// TIA Portal V19 export
FUNCTION_BLOCK "CoilHandling_FB"   // FB101, LAD
TITLE = COIL HANDLING MANAGER
// stored: MemoryReserve 100, SetENOAutomatically false
   VAR_INPUT
      AreaInterface : "AreaInterface";
      ZSI : "udt_ZoneSafetyInterface";
      DataIn : Struct
         PbMaterialBkw : Bool;
         PbMaterialFwd : Bool;
         PbExtraLowSpeed : Bool;
         SensorMatPresence_Decoiler : Bool;
         SensorMatPresence_StraightEntry : Bool;
         SensorMatPresence_StraightExit : Bool;
         SensorMatPresence_JBPinchExit : Bool;
         PbCoilReady : Bool;
         PbProvino : Bool;
         Decoiler2_PosizioneRazza : Bool;
      END_STRUCT;
      CIn : Struct
         DecoilersHRot : "DecoilersHRot_Status";
         Decoiler1 : "Decoiler_Status";
         Decoiler2 : "Decoiler_Status";
         Peeler : "Peeler_Status";
         Straigtener : "Straightener_Status";
         JB : "JB_Status";
         MaterialCounter : Struct
            AlrPresence : Bool;
            WngPresence : Bool;
            Data : "MatCountData";
         END_STRUCT;
         Loop : Struct
            SystemOn : Bool;
            Enable_FWD : Bool;
            Enable_BWD : Bool;
            SynchroRunning : Bool;
            MaxLength_Reeached : Bool;
            VelocityOverride : Real;
         END_STRUCT;
         Downstream : Struct
            Aut : Bool;
            MaterialPresence_Entry : Bool;
            MaterialPresence : Bool;
            LineVelocity : LReal;
         END_STRUCT;
         MES : "Prod_Coil_Ctrl";
      END_STRUCT;
      Config : "CoilHandling_Config";
      "ThicknessCheck_HW_ID_DL-PN" : HW_SUBMODULE := 784;
      ThicknessCheck_HW_ID_IL1000 : HW_SUBMODULE := 1042;
      ThicknessCheck_HW_ID_IL1050 : HW_SUBMODULE := 1043;
   END_VAR
   VAR_OUTPUT
      MachineInterface : "MachineInterface";
      COut : Struct
         Gen : Struct
            Material_STS : Int;   // 0=Empty; 1=Threading; 2= Full; 3= EOF Coil; 4= Separation
            MaterialPresence : Bool;
            MaterialMissing : Bool;
            NextEndOfMaterial : Bool;
            EmptyingConfirmed : Bool := FALSE;
            ExtraLowSpeedSelection : Bool;
            SemiAutomatic : Bool;
            Production_Running : Bool;
            DecoilerInLineNumber : Int;
            CoilDiameter : Real;
         END_STRUCT;
         DecoilersHRot : "DecoilersHRot_Manager";
         DecoilerInLine : "Decoiler_Manager";
         DecoilerOutLine : "Decoiler_Manager";
         Decoiler1 : "Decoiler_Manager";
         Decoiler2 : "Decoiler_Manager";
         Peeler : "Peeler_Manager";
         Straightener : "Straightener_Manager";
         JB : "JB_Manager";
         Loop : Struct
            Stop : Bool;
            Synchro_Request : Bool;
            MaterialMiddlePos_Request : Bool;
         END_STRUCT;
         MES : Struct
            Deroga_Spessore_Errato { ExternalWritable := 'False'} : Bool;
            Spessore_Lamiera_Errato { ExternalWritable := 'False'} : Bool;
            Spessore_Lamiera_Sensore_Valore : Real;
            Spessore_Lamiera_Errore_Valore { ExternalWritable := 'False'} : Real;
            Provino_Eseguito : Bool;
         END_STRUCT;
      END_STRUCT;
      DataOut : Struct
         Lamp_CoilReady : Bool;
         Lamp_ExtraLowSpeed : Bool;
         Lamp_Provino : Bool;
      END_STRUCT;
   END_VAR
   VAR_IN_OUT
      Pers : "CoilHandling_Persistent";
   END_VAR
   VAR
      Alarm : Struct
         MaterialMissing : Bool;
         S_MatPresence_StraightExit_NotOFF : Bool;
         MatCounterAlrPresence : Bool;
         EndOfMaterial : Bool;
         TichnessCheck { ExternalAccessible := 'False'; ExternalVisible := 'False'; ExternalWritable := 'False'} : Struct
            Err_Sensor_Get_PN_IO : Bool;
            Err_Sensor_Rack : Bool;
            Err_Sensor_Value : Bool;
            ThicknessOutOfRange : Bool;
         END_STRUCT;
         MES : Struct
            STOP_Provino { ExternalAccessible := 'False'; ExternalVisible := 'False'; ExternalWritable := 'False'} : Bool;
            STOP_Taglio_Fine_Ordini { ExternalAccessible := 'False'; ExternalVisible := 'False'; ExternalWritable := 'False'} : Bool;
            STOP_Manca_Dati_AspoInLinea { ExternalAccessible := 'False'; ExternalVisible := 'False'; ExternalWritable := 'False'} : Bool;
            STOP_FineTurno { ExternalAccessible := 'False'; ExternalVisible := 'False'; ExternalWritable := 'False'} : Bool;
            STOP_ControlloQualita { ExternalAccessible := 'False'; ExternalVisible := 'False'; ExternalWritable := 'False'} : Bool;
         END_STRUCT;
      END_STRUCT;
      Warning : Struct
         NotAutReady : Bool;
         MatCounterWngPresence : Bool;
         EmptyingIsON : Bool := FALSE;
         EndOfMaterial_StraightenetEntry : Bool;
         EndOfMaterial_StraightenetExit : Bool;
         EndOfCoilSequenceRunning : Bool;
         ExtraLowSpeedIsON : Bool;
         Decoiler2_RazzaNonInPosizione : Bool;
         StopInactivity : Bool;
         ThicnessCheck { ExternalAccessible := 'False'; ExternalVisible := 'False'; ExternalWritable := 'False'} : Struct
            SensorDisable : Bool;
            ThicknessOutOfRange : Bool;
            Err_Bypass : Bool;
         END_STRUCT;
         MES : Struct
            STOP_Manca_Dati_AspoInCarico : Bool;
         END_STRUCT;
      END_STRUCT;
      HMI : Struct
         B_ConfirmEmptying { ExternalAccessible := 'False'; ExternalVisible := 'False'; ExternalWritable := 'False'} : Bool;
         B_ConfirmEmptyingShow { ExternalAccessible := 'False'; ExternalVisible := 'False'; ExternalWritable := 'False'} : Bool;
         B_ConfirmEmptyingStatus : Bool;
         ThicknessControl : Struct
            Button_Exception : Bool;
            Button_Init : Bool;
            STATUS : Int;
         END_STRUCT;
      END_STRUCT;
      Ctrl : Struct
         Pause : Bool;
         Stop : Bool;
         Semiautomatic_MaterialFwd : Bool;
         Semiautomatic_MaterialBkw : Bool;
         EndOfCoil : Struct
            StraightRollEntry_Open : Bool;
            StraightRollExit_Open : Bool;
            StraightRollEntry_Close : Bool;
            StraightRollExit_Close : Bool;
            Straightener_Bwd : Bool;
            Straightener_Fwd : Bool;
            JB_Pinch_Open : Bool;
            JB_Pinch_Close : Bool;
            JB_Pinch_Fwd : Bool;
            JB_Cut_Rest : Bool;
            JB_Cut_Work : Bool;
            JB_Welder_Open : Bool;
            TargetPosMat_StraightEmpty : LReal;
            TargetPosMat_TailCutExe : LReal;
            TargetPosMat_JunctionExe : LReal;
            ChangeCoilExe : Bool;
            Decoiler_Fwd : Bool;
         END_STRUCT;
      END_STRUCT;
      Sts : Struct
         FeedStandstill : Bool;
         AlarmsPresence : Bool;
         WarningsPresence : Bool;
         EnableCycleStopProgrammed : Bool;
         MaterialFwdEnable : Bool;
         MaterialBkwEnable : Bool;
         CumulativeMaterialFwdRequest : Bool;
         Semiautomatic : Bool;
         ExtraLowSpeedSelectionPB : Bool;
         ExtraLowSpeedSelection : Bool;
         STOP_Feed_by_MES : Bool;
         STOP_CoilChange_By_MES : Bool;
         STOP_Inactivity : Bool;
         DecoilerInLine : "Decoiler_Status";
         DecoilerOutOfLine : "Decoiler_Status";
         EndOfCoil : Struct
            Status : Int;
            Cnd : Bool;
            Idle : Bool;
            EndOfSequence : Bool;
            PinchRoll_SpaceToStop : LReal;
            PosMat_AtEndMatPresence_StraightEnty : LReal;
            PosMat_AtEndMatPresence_StraightExit : LReal;
            MissingTargetPosMat_StraightEmpty : LReal;
            MissingToTargetPosMat_TailCutExe : LReal;
            StopPinchRoll_TargetPosMat_TailCutExe : Bool;
            Reached_TargetPosMat_TailCutExe : Bool;
            MissingToTargetPosMat_JunctionExe : LReal;
            StopPinchRoll_TargetPosMat_JunctionExe : Bool;
            Reached_TargetPosMat_JunctionExe : Bool;
         END_STRUCT;
         LoopSynchro : Struct
            Phase1_A : Bool;   // Coil diameter < limit
            Phase2_A : Bool;   // Mem synchro done
            Phase1_B : Bool;   // Coil diameter < limit
            Phase2_B : Bool;   // Mem synchro done
         END_STRUCT;
         MaterialMoveSemiAut : Struct
            Bwd_Phase1 : Bool;   // Move no feeding machine to rest
            Bwd_Phase1Cnd : Bool;
            Bwd_Phase2 : Bool;   // Move velocity = 0
            Bwd_Phase2Cnd : Bool;
            Bwd_Phase3 : Bool;   // Move velocity > 0
            Fwd_Phase1 : Bool;   // Move no feeding machine to rest
            Fwd_Phase1Cnd : Bool;
            Fwd_Phase2 : Bool;   // Move velocity = 0
            Fwd_Phase2Cnd : Bool;
            Fwd_Phase3 : Bool;   // Move velocity > 0
         END_STRUCT;
         MaterialMoveAut : Struct
            Fwd_Phase1 : Bool;   // Move no feeding machine to rest
            Fwd_Phase1Cnd : Bool;
            Fwd_Phase2 : Bool;   // Move velocity = 0
            Fwd_Phase2Cnd : Bool;
            Fwd_Phase3 : Bool;   // Move velocity > 0
         END_STRUCT;
      END_STRUCT;
      MatPresence_Decoiler : "DelayOnOff_R";
      MatPresence_StraightEntry : "DelayOnOff_R";
      MatPresence_StraightExit : "DelayOnOff_R";
      MatPresence_JBPinchExit : "DelayOnOff_R";
      Coil_LooseWrap : "CoilCheckLooseWrap";
      ThicknessCheck { S7_SetPoint := 'True'} : "ThicknessCheck_FB";
      CoilHandling_MES { S7_SetPoint := 'True'} : "CoilHandling_MES_FB";
      TON_Emptying : TON_TIME;
      TON_DecoilerNotMovingBkw : TON_TIME;
      TON_PinchrollFwd : TON_TIME;
      TON_StraightnerBwd : TON_TIME;
      TON_StraightnerFwd : TON_TIME;
      TON_SemiautoOFF : TON_TIME;
      TON_AutDisableAxes : TON_TIME;
      TON_StopInactivity : TON_TIME;
      AUX : Struct
         S_MatPresence_StraightEntry : Bool;
         S_MatPresence_StraightExit : Bool;
         PbMaterialFwd : Bool;
         PbMaterialBkw : Bool;
         PbExtraLowSpeed : Bool;
         ButtonForceLoopMiddle : Bool;
         PbCoilLoaded : Bool;
         StopLoop { ExternalAccessible := 'False'; ExternalVisible := 'False'; ExternalWritable := 'False'} : Bool;
      END_STRUCT;
   END_VAR
   VAR_TEMP
      PE : Struct
         Not_S_MatPresence_StraightEntry : Bool;
         Not_S_MatPresence_StraightExit : Bool;
         PbMaterialBkw : Bool;
         PbMaterialFwd : Bool;
         PbExtraLowSpeed : Bool;
      END_STRUCT;
      Req : Bool;
      Set : Bool;
      Rst : Bool;
      Cnd : Bool;
      Min : Bool;
      Max : Bool;
      OK : Bool;
      StraightRollEntry_Used : Bool;
      StraightRollExit_Used : Bool;
      DistanceSensorEntryExitStraight : LReal;
      DistanceLimit : LReal;
      LineVel : LReal;
      Decoiler_VelFactor : LReal;
      Straightener_VelFactor : LReal;
      OverRide_VelFactor : LReal;
      OverRide_VelFactor_Candidate : LReal;
      Delta : LReal;
      Vel : LReal;
      EnableStopInPhase : Bool;
      EnableStopProgrammed : Bool;
      EnableStopDoorOpeningReq : Bool;
      Set_1 : Bool;
      Rst_1 : Bool;
      Set_2 : Bool;
      Rst_2 : Bool;
      CaseA : Bool;
      CaseB : Bool;
      Empty : Bool;
      JunctionDone : Bool;
   END_VAR
   // MachineInterface.AutReady := TRUE;
   // MachineInterface.Aborting := FALSE;
   // MachineInterface.AckStopInPhase := FALSE;
   // MachineInterface.AckStopProgrammed := FALSE;
   // MachineInterface.MotionsStandStill := TRUE;
   // MachineInterface.AlarmsPresence := FALSE;
   // MachineInterface.WarningPresence := TRUE;
   VAR_TEMP   // added for the SCL form of the ladder/FBD networks
      _w1 : Bool;
      _w2 : Bool;
      _w3 : Bool;
   END_VAR
BEGIN

REGION Network 1 (SCL): Reset alarms
   IF #AreaInterface.RstAlarms THEN

       #Alarm.MaterialMissing := FALSE;
       #Alarm.S_MatPresence_StraightExit_NotOFF := FALSE;
       #Alarm.EndOfMaterial := FALSE;


       #Warning.Decoiler2_RazzaNonInPosizione := FALSE;
       #Warning.NotAutReady := FALSE;

   END_IF;
END_REGION

REGION Network 2: >
END_REGION

REGION Network 3: >
END_REGION

REGION Network 4: Straightenetr rolls entry / exit to use
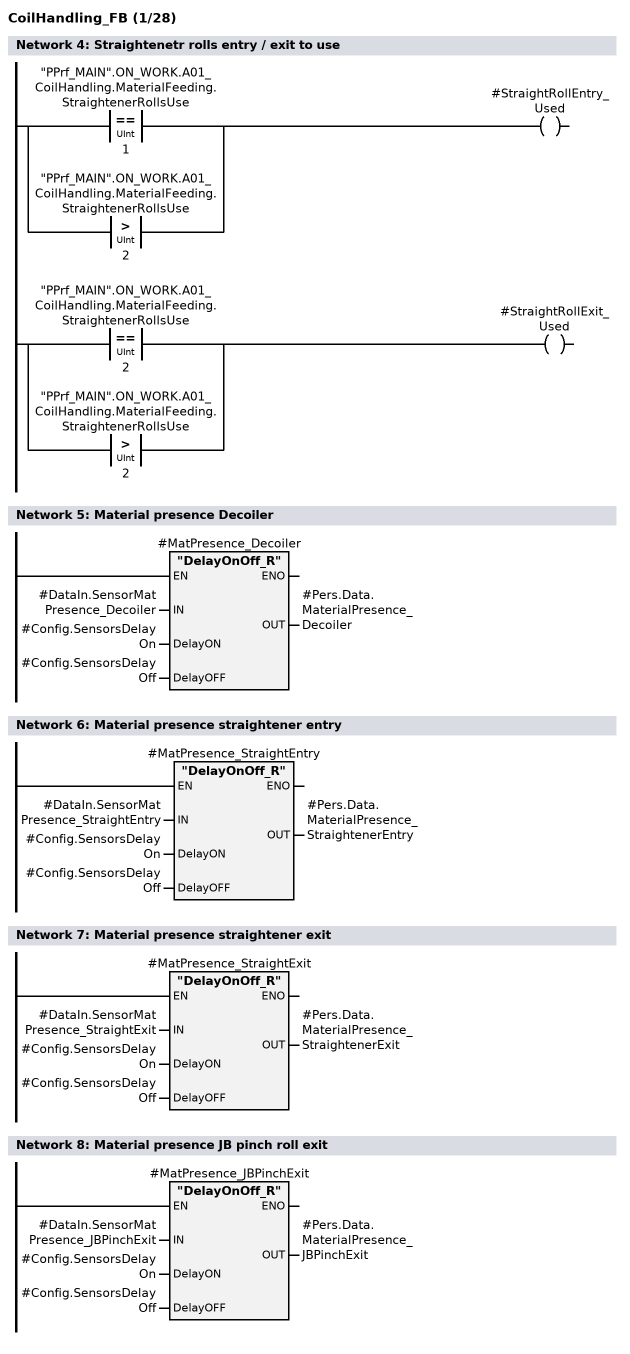
   RUNG wire#powerrail
      { S7_Templates := "SrcType := UInt" } EQ_Contact(in1 := "PPrf_MAIN".ON_WORK.A01_CoilHandling.MaterialFeeding.StraightenerRollsUse, in2 := 1)
      wire#w1
      Coil( #StraightRollEntry_Used )
   END_RUNG
   RUNG wire#powerrail
      { S7_Templates := "SrcType := UInt" } GT_Contact(in1 := "PPrf_MAIN".ON_WORK.A01_CoilHandling.MaterialFeeding.StraightenerRollsUse, in2 := 2)
   END_RUNG wire#w1
   RUNG wire#powerrail
      { S7_Templates := "SrcType := UInt" } EQ_Contact(in1 := "PPrf_MAIN".ON_WORK.A01_CoilHandling.MaterialFeeding.StraightenerRollsUse, in2 := 2)
      wire#w2
      Coil( #StraightRollExit_Used )
   END_RUNG
   RUNG wire#powerrail
      { S7_Templates := "SrcType := UInt" } GT_Contact(in1 := "PPrf_MAIN".ON_WORK.A01_CoilHandling.MaterialFeeding.StraightenerRollsUse, in2 := 2)
   END_RUNG wire#w2
   // the same network as SCL:
   #StraightRollEntry_Used := ("PPrf_MAIN".ON_WORK.A01_CoilHandling.MaterialFeeding.StraightenerRollsUse = 1) OR ("PPrf_MAIN".ON_WORK.A01_CoilHandling.MaterialFeeding.StraightenerRollsUse > 2);
   #StraightRollExit_Used := ("PPrf_MAIN".ON_WORK.A01_CoilHandling.MaterialFeeding.StraightenerRollsUse = 2) OR ("PPrf_MAIN".ON_WORK.A01_CoilHandling.MaterialFeeding.StraightenerRollsUse > 2);
END_REGION

REGION Network 5: Material presence Decoiler
   RUNG wire#powerrail
      #MatPresence_Decoiler(IN := #DataIn.SensorMatPresence_Decoiler, DelayON := #Config.SensorsDelayOn, DelayOFF := #Config.SensorsDelayOff, OUT => #Pers.Data.MaterialPresence_Decoiler)
   END_RUNG
   // the same network as SCL:
   #MatPresence_Decoiler(IN := #DataIn.SensorMatPresence_Decoiler,   // "DelayOnOff_R"
                         DelayON := #Config.SensorsDelayOn,
                         DelayOFF := #Config.SensorsDelayOff,
                         OUT => #Pers.Data.MaterialPresence_Decoiler);
END_REGION

REGION Network 6: Material presence straightener entry
   RUNG wire#powerrail
      #MatPresence_StraightEntry(IN := #DataIn.SensorMatPresence_StraightEntry, DelayON := #Config.SensorsDelayOn, DelayOFF := #Config.SensorsDelayOff, OUT => #Pers.Data.MaterialPresence_StraightenerEntry)
   END_RUNG
   // the same network as SCL:
   #MatPresence_StraightEntry(IN := #DataIn.SensorMatPresence_StraightEntry,   // "DelayOnOff_R"
                           DelayON := #Config.SensorsDelayOn,
                           DelayOFF := #Config.SensorsDelayOff,
                           OUT => #Pers.Data.MaterialPresence_StraightenerEntry);
END_REGION

REGION Network 7: Material presence straightener exit
   RUNG wire#powerrail
      #MatPresence_StraightExit(IN := #DataIn.SensorMatPresence_StraightExit, DelayON := #Config.SensorsDelayOn, DelayOFF := #Config.SensorsDelayOff, OUT => #Pers.Data.MaterialPresence_StraightenerExit)
   END_RUNG
   // the same network as SCL:
   #MatPresence_StraightExit(IN := #DataIn.SensorMatPresence_StraightExit,   // "DelayOnOff_R"
                           DelayON := #Config.SensorsDelayOn,
                           DelayOFF := #Config.SensorsDelayOff,
                           OUT => #Pers.Data.MaterialPresence_StraightenerExit);
END_REGION

REGION Network 8: Material presence JB pinch roll exit
   RUNG wire#powerrail
      #MatPresence_JBPinchExit(IN := #DataIn.SensorMatPresence_JBPinchExit, DelayON := #Config.SensorsDelayOn, DelayOFF := #Config.SensorsDelayOff, OUT => #Pers.Data.MaterialPresence_JBPinchExit)
   END_RUNG
   // the same network as SCL:
   #MatPresence_JBPinchExit(IN := #DataIn.SensorMatPresence_JBPinchExit,   // "DelayOnOff_R"
                           DelayON := #Config.SensorsDelayOn,
                           DelayOFF := #Config.SensorsDelayOff,
                           OUT => #Pers.Data.MaterialPresence_JBPinchExit);
END_REGION

REGION Network 9: >
END_REGION

REGION Network 10: >
END_REGION

REGION Network 11: Material junction done
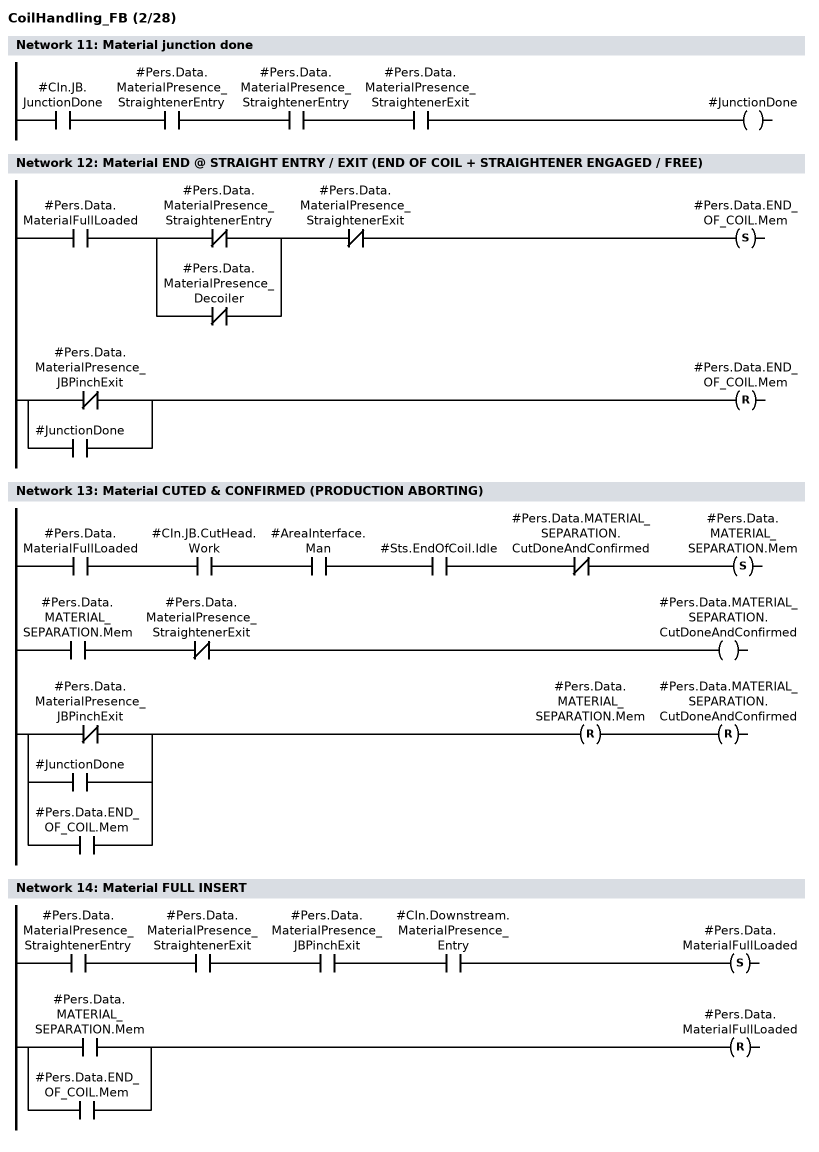
   RUNG wire#powerrail
      Contact( #CIn.JB.JunctionDone )
      Contact( #Pers.Data.MaterialPresence_StraightenerEntry )
      Contact( #Pers.Data.MaterialPresence_StraightenerEntry )
      Contact( #Pers.Data.MaterialPresence_StraightenerExit )
      Coil( #JunctionDone )
   END_RUNG
   // the same network as SCL:
   #JunctionDone := #CIn.JB.JunctionDone AND #Pers.Data.MaterialPresence_StraightenerEntry AND #Pers.Data.MaterialPresence_StraightenerEntry AND #Pers.Data.MaterialPresence_StraightenerExit;
END_REGION

REGION Network 12: Material END @ STRAIGHT ENTRY / EXIT (END OF COIL + STRAIGHTENER ENGAGED / FREE)
   RUNG wire#powerrail
      Contact( #Pers.Data.MaterialFullLoaded )
      wire#w1
      I_Contact( #Pers.Data.MaterialPresence_StraightenerEntry )
      wire#w2
      I_Contact( #Pers.Data.MaterialPresence_StraightenerExit )
      S_Coil( #Pers.Data.END_OF_COIL.Mem )
   END_RUNG
   RUNG wire#w1
      I_Contact( #Pers.Data.MaterialPresence_Decoiler )
   END_RUNG wire#w2
   RUNG wire#powerrail
      I_Contact( #Pers.Data.MaterialPresence_JBPinchExit )
      wire#w3
      R_Coil( #Pers.Data.END_OF_COIL.Mem )
   END_RUNG
   RUNG wire#powerrail
      Contact( #JunctionDone )
   END_RUNG wire#w3
   // the same network as SCL:
   IF #Pers.Data.MaterialFullLoaded AND (NOT #Pers.Data.MaterialPresence_StraightenerEntry OR NOT #Pers.Data.MaterialPresence_Decoiler) AND NOT #Pers.Data.MaterialPresence_StraightenerExit THEN
       #Pers.Data.END_OF_COIL.Mem := TRUE;
   END_IF;
   IF NOT #Pers.Data.MaterialPresence_JBPinchExit OR #JunctionDone THEN
       #Pers.Data.END_OF_COIL.Mem := FALSE;
   END_IF;
END_REGION

REGION Network 13: Material CUTED & CONFIRMED (PRODUCTION ABORTING)
   RUNG wire#powerrail
      Contact( #Pers.Data.MaterialFullLoaded )
      Contact( #CIn.JB.CutHead.Work )
      Contact( #AreaInterface.Man )
      Contact( #Sts.EndOfCoil.Idle )
      I_Contact( #Pers.Data.MATERIAL_SEPARATION.CutDoneAndConfirmed )
      S_Coil( #Pers.Data.MATERIAL_SEPARATION.Mem )
   END_RUNG
   RUNG wire#powerrail
      Contact( #Pers.Data.MATERIAL_SEPARATION.Mem )
      I_Contact( #Pers.Data.MaterialPresence_StraightenerExit )
      Coil( #Pers.Data.MATERIAL_SEPARATION.CutDoneAndConfirmed )
   END_RUNG
   RUNG wire#powerrail
      I_Contact( #Pers.Data.MaterialPresence_JBPinchExit )
      wire#w1
      R_Coil( #Pers.Data.MATERIAL_SEPARATION.Mem )
      R_Coil( #Pers.Data.MATERIAL_SEPARATION.CutDoneAndConfirmed )
   END_RUNG
   RUNG wire#powerrail
      Contact( #JunctionDone )
   END_RUNG wire#w1
   RUNG wire#powerrail
      Contact( #Pers.Data.END_OF_COIL.Mem )
   END_RUNG wire#w1
   // the same network as SCL:
   IF #Pers.Data.MaterialFullLoaded AND #CIn.JB.CutHead.Work AND #AreaInterface.Man AND #Sts.EndOfCoil.Idle AND NOT #Pers.Data.MATERIAL_SEPARATION.CutDoneAndConfirmed THEN
       #Pers.Data.MATERIAL_SEPARATION.Mem := TRUE;
   END_IF;
   #Pers.Data.MATERIAL_SEPARATION.CutDoneAndConfirmed := #Pers.Data.MATERIAL_SEPARATION.Mem AND NOT #Pers.Data.MaterialPresence_StraightenerExit;
   IF NOT #Pers.Data.MaterialPresence_JBPinchExit OR #JunctionDone OR #Pers.Data.END_OF_COIL.Mem THEN
       #Pers.Data.MATERIAL_SEPARATION.Mem := FALSE;
       #Pers.Data.MATERIAL_SEPARATION.CutDoneAndConfirmed := FALSE;
   END_IF;
END_REGION

REGION Network 14: Material FULL INSERT
   RUNG wire#powerrail
      Contact( #Pers.Data.MaterialPresence_StraightenerEntry )
      Contact( #Pers.Data.MaterialPresence_StraightenerExit )
      Contact( #Pers.Data.MaterialPresence_JBPinchExit )
      Contact( #CIn.Downstream.MaterialPresence_Entry )
      S_Coil( #Pers.Data.MaterialFullLoaded )
   END_RUNG
   RUNG wire#powerrail
      Contact( #Pers.Data.MATERIAL_SEPARATION.Mem )
      wire#w1
      R_Coil( #Pers.Data.MaterialFullLoaded )
   END_RUNG
   RUNG wire#powerrail
      Contact( #Pers.Data.END_OF_COIL.Mem )
   END_RUNG wire#w1
   // the same network as SCL:
   IF #Pers.Data.MaterialPresence_StraightenerEntry AND #Pers.Data.MaterialPresence_StraightenerExit AND #Pers.Data.MaterialPresence_JBPinchExit AND #CIn.Downstream.MaterialPresence_Entry THEN
       #Pers.Data.MaterialFullLoaded := TRUE;
   END_IF;
   IF #Pers.Data.MATERIAL_SEPARATION.Mem OR #Pers.Data.END_OF_COIL.Mem THEN
       #Pers.Data.MaterialFullLoaded := FALSE;
   END_IF;
END_REGION

REGION Network 15: Material presence for keep running the material even thoug is not full insterted
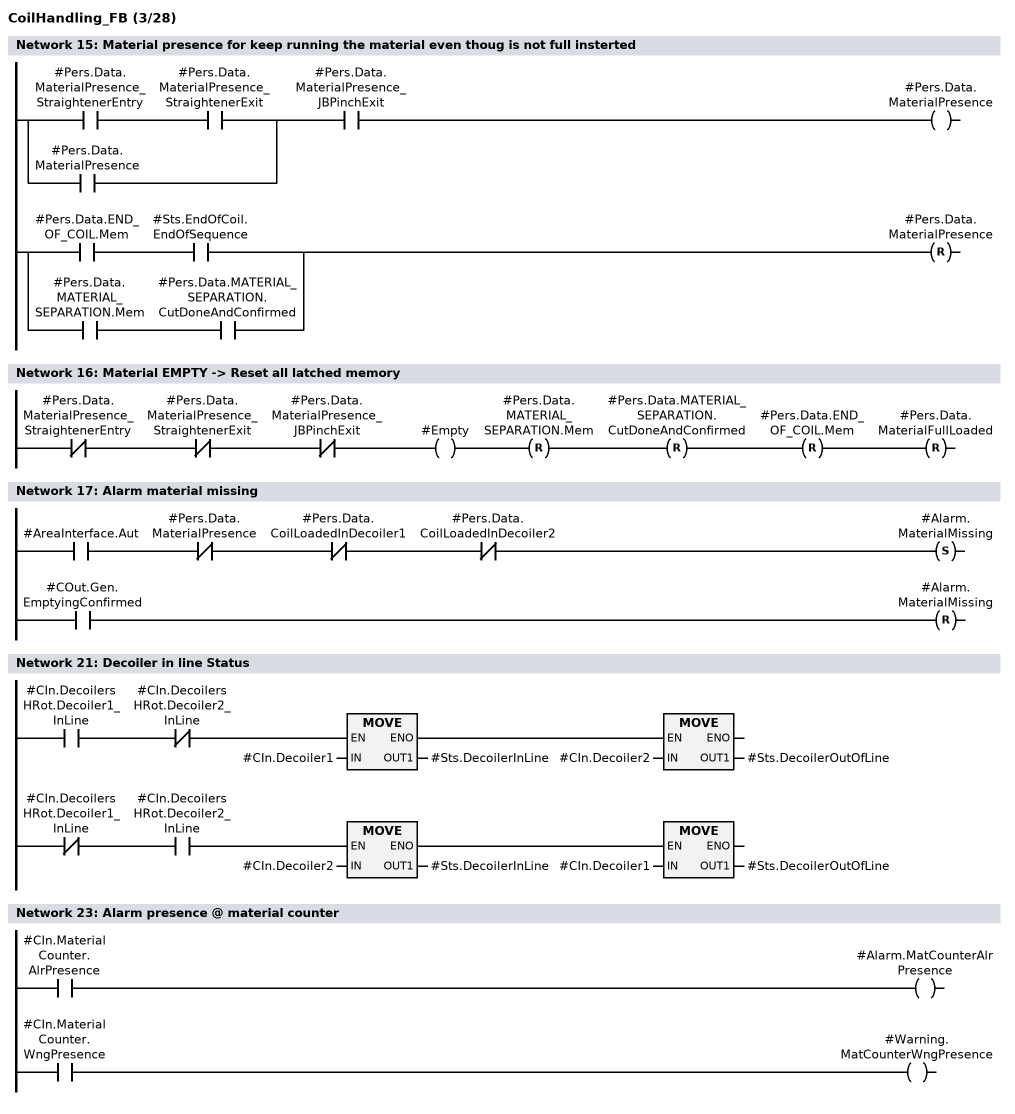
   RUNG wire#powerrail
      Contact( #Pers.Data.MaterialPresence_StraightenerEntry )
      Contact( #Pers.Data.MaterialPresence_StraightenerExit )
      wire#w1
      Contact( #Pers.Data.MaterialPresence_JBPinchExit )
      Coil( #Pers.Data.MaterialPresence )
   END_RUNG
   RUNG wire#powerrail
      Contact( #Pers.Data.MaterialPresence )
   END_RUNG wire#w1
   RUNG wire#powerrail
      Contact( #Pers.Data.END_OF_COIL.Mem )
      Contact( #Sts.EndOfCoil.EndOfSequence )
      wire#w2
      R_Coil( #Pers.Data.MaterialPresence )
   END_RUNG
   RUNG wire#powerrail
      Contact( #Pers.Data.MATERIAL_SEPARATION.Mem )
      Contact( #Pers.Data.MATERIAL_SEPARATION.CutDoneAndConfirmed )
   END_RUNG wire#w2
   // the same network as SCL:
   #Pers.Data.MaterialPresence := ((#Pers.Data.MaterialPresence_StraightenerEntry AND #Pers.Data.MaterialPresence_StraightenerExit) OR #Pers.Data.MaterialPresence) AND #Pers.Data.MaterialPresence_JBPinchExit;
   IF (#Pers.Data.END_OF_COIL.Mem AND #Sts.EndOfCoil.EndOfSequence) OR (#Pers.Data.MATERIAL_SEPARATION.Mem AND #Pers.Data.MATERIAL_SEPARATION.CutDoneAndConfirmed) THEN
       #Pers.Data.MaterialPresence := FALSE;
   END_IF;
END_REGION

REGION Network 16: Material EMPTY -> Reset all latched memory
   RUNG wire#powerrail
      I_Contact( #Pers.Data.MaterialPresence_StraightenerEntry )
      I_Contact( #Pers.Data.MaterialPresence_StraightenerExit )
      I_Contact( #Pers.Data.MaterialPresence_JBPinchExit )
      Coil( #Empty )
      R_Coil( #Pers.Data.MATERIAL_SEPARATION.Mem )
      R_Coil( #Pers.Data.MATERIAL_SEPARATION.CutDoneAndConfirmed )
      R_Coil( #Pers.Data.END_OF_COIL.Mem )
      R_Coil( #Pers.Data.MaterialFullLoaded )
   END_RUNG
   // the same network as SCL:
   #Empty := NOT #Pers.Data.MaterialPresence_StraightenerEntry AND NOT #Pers.Data.MaterialPresence_StraightenerExit AND NOT #Pers.Data.MaterialPresence_JBPinchExit;
   IF #Empty THEN
       #Pers.Data.MATERIAL_SEPARATION.Mem := FALSE;
       #Pers.Data.MATERIAL_SEPARATION.CutDoneAndConfirmed := FALSE;
       #Pers.Data.END_OF_COIL.Mem := FALSE;
       #Pers.Data.MaterialFullLoaded := FALSE;
   END_IF;
END_REGION

REGION Network 17: Alarm material missing
   RUNG wire#powerrail
      Contact( #AreaInterface.Aut )
      I_Contact( #Pers.Data.MaterialPresence )
      I_Contact( #Pers.Data.CoilLoadedInDecoiler1 )
      I_Contact( #Pers.Data.CoilLoadedInDecoiler2 )
      S_Coil( #Alarm.MaterialMissing )
   END_RUNG
   RUNG wire#powerrail
      Contact( #COut.Gen.EmptyingConfirmed )
      R_Coil( #Alarm.MaterialMissing )
   END_RUNG
   // the same network as SCL:
   IF #AreaInterface.Aut AND NOT #Pers.Data.MaterialPresence AND NOT #Pers.Data.CoilLoadedInDecoiler1 AND NOT #Pers.Data.CoilLoadedInDecoiler2 THEN
       #Alarm.MaterialMissing := TRUE;
   END_IF;
   IF #COut.Gen.EmptyingConfirmed THEN #Alarm.MaterialMissing := FALSE; END_IF;
END_REGION

REGION Network 18: >
END_REGION

REGION Network 19 (SCL): Material status
   IF #Empty
   THEN
       #COut.Gen.Material_STS := "MAT_EMPTY";
   ELSIF #Pers.Data.END_OF_COIL.Mem
   THEN
       #COut.Gen.Material_STS := "MAT_EOF_COIL";
   ELSIF #Pers.Data.MATERIAL_SEPARATION.Mem
   THEN
       #COut.Gen.Material_STS := "MAT_SPERATION";

   ELSIF #Pers.Data.MaterialFullLoaded
   THEN
       #COut.Gen.Material_STS := "MAT_FULL";
   ELSE
       #COut.Gen.Material_STS := "MAT_INTRODUCTION";
   END_IF;
END_REGION

REGION Network 20: >
END_REGION

REGION Network 21: Decoiler in line Status
   RUNG wire#powerrail
      Contact( #CIn.DecoilersHRot.Decoiler1_InLine )
      I_Contact( #CIn.DecoilersHRot.Decoiler2_InLine )
      Move(in := #CIn.Decoiler1, out1 => #Sts.DecoilerInLine)
      Move(in := #CIn.Decoiler2, out1 => #Sts.DecoilerOutOfLine)
   END_RUNG
   RUNG wire#powerrail
      I_Contact( #CIn.DecoilersHRot.Decoiler1_InLine )
      Contact( #CIn.DecoilersHRot.Decoiler2_InLine )
      Move(in := #CIn.Decoiler2, out1 => #Sts.DecoilerInLine)
      Move(in := #CIn.Decoiler1, out1 => #Sts.DecoilerOutOfLine)
   END_RUNG
   // the same network as SCL:
   IF #CIn.DecoilersHRot.Decoiler1_InLine AND NOT #CIn.DecoilersHRot.Decoiler2_InLine THEN
       #Sts.DecoilerInLine := #CIn.Decoiler1;
       #Sts.DecoilerOutOfLine := #CIn.Decoiler2;
   END_IF;
   IF NOT #CIn.DecoilersHRot.Decoiler1_InLine AND #CIn.DecoilersHRot.Decoiler2_InLine THEN
       #Sts.DecoilerInLine := #CIn.Decoiler2;
       #Sts.DecoilerOutOfLine := #CIn.Decoiler1;
   END_IF;
END_REGION

REGION Network 22: >
END_REGION

REGION Network 23: Alarm presence @ material counter
   RUNG wire#powerrail
      Contact( #CIn.MaterialCounter.AlrPresence )
      Coil( #Alarm.MatCounterAlrPresence )
   END_RUNG
   RUNG wire#powerrail
      Contact( #CIn.MaterialCounter.WngPresence )
      Coil( #Warning.MatCounterWngPresence )
   END_RUNG
   // the same network as SCL:
   #Alarm.MatCounterAlrPresence := #CIn.MaterialCounter.AlrPresence;
   #Warning.MatCounterWngPresence := #CIn.MaterialCounter.WngPresence;
END_REGION

REGION Network 24: >
END_REGION

REGION Network 25: >
END_REGION

REGION Network 26: Area Emptying
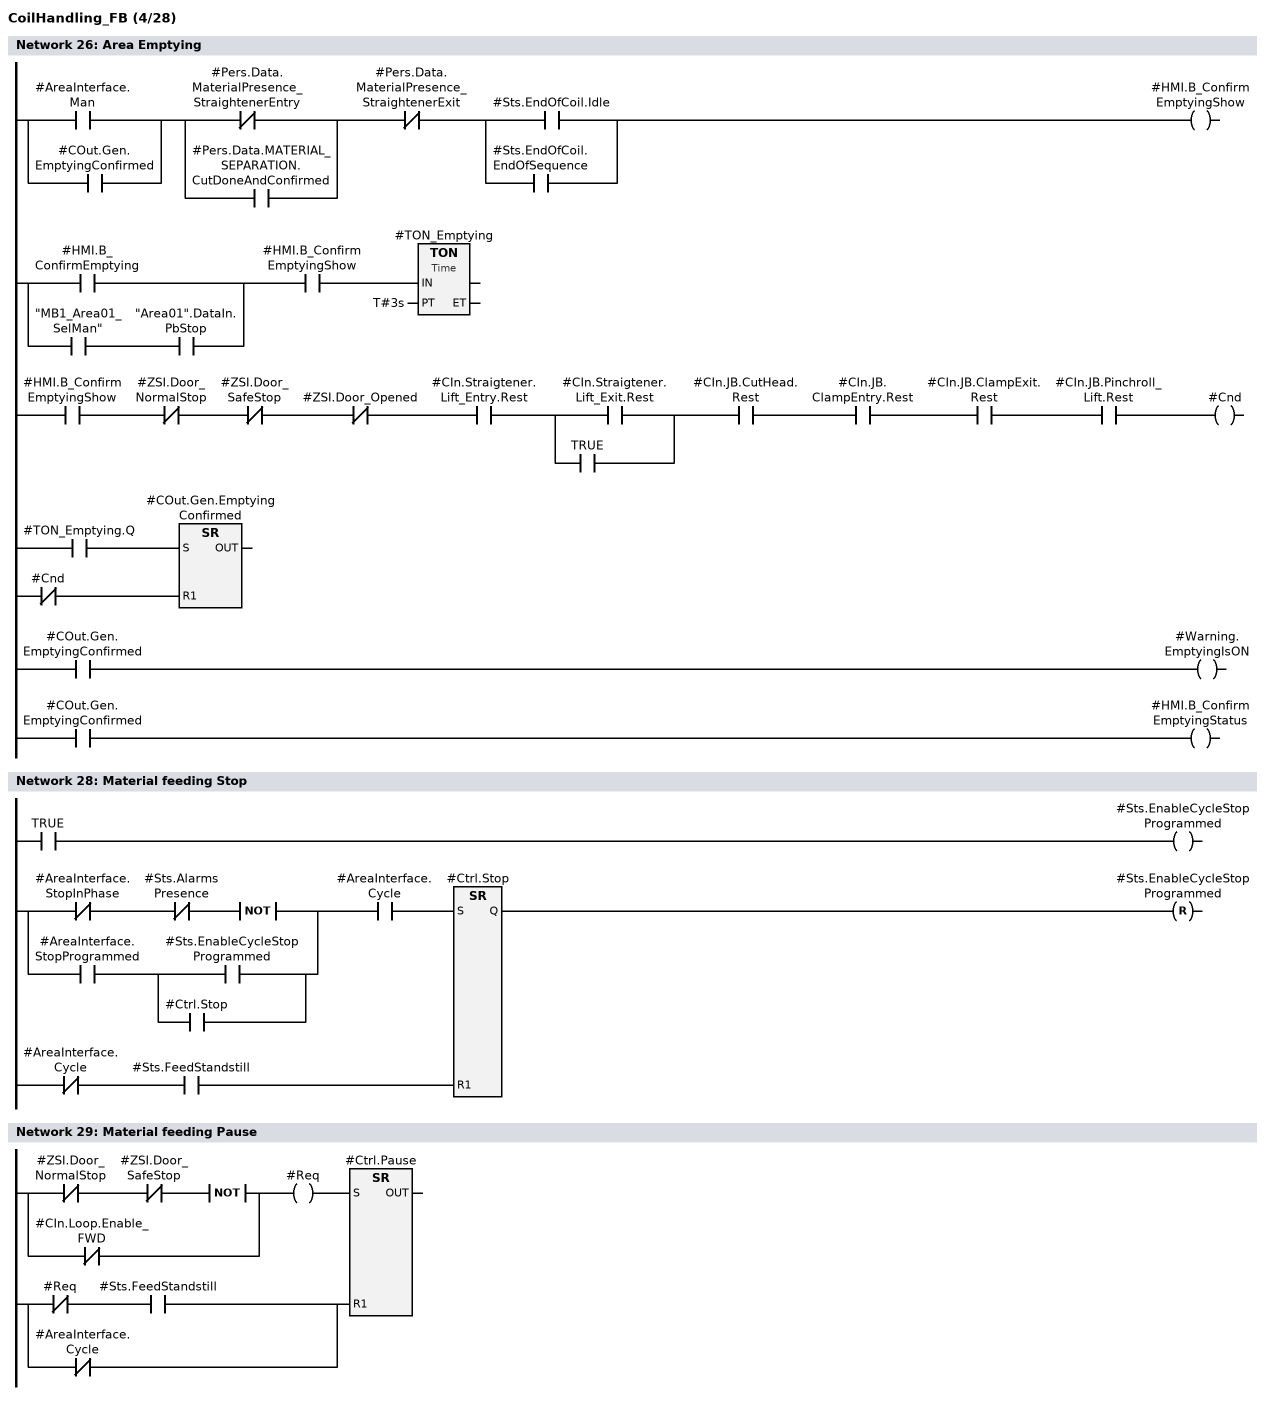
   RUNG wire#powerrail
      Contact( #AreaInterface.Man )
      wire#w1
      I_Contact( #Pers.Data.MaterialPresence_StraightenerEntry )
      wire#w2
      I_Contact( #Pers.Data.MaterialPresence_StraightenerExit )
      wire#w3
      Contact( #Sts.EndOfCoil.Idle )
      wire#w4
      Coil( #HMI.B_ConfirmEmptyingShow )
   END_RUNG
   RUNG wire#powerrail
      Contact( #COut.Gen.EmptyingConfirmed )
   END_RUNG wire#w1
   RUNG wire#w1
      Contact( #Pers.Data.MATERIAL_SEPARATION.CutDoneAndConfirmed )
   END_RUNG wire#w2
   RUNG wire#w3
      Contact( #Sts.EndOfCoil.EndOfSequence )
   END_RUNG wire#w4
   RUNG wire#powerrail
      Contact( #HMI.B_ConfirmEmptying )
      wire#w5
      Contact( #HMI.B_ConfirmEmptyingShow )
      { S7_Templates := "time_type := Time" } #TON_Emptying.TON(pt := T#3s, et =>)
   END_RUNG
   RUNG wire#powerrail
      Contact( "MB1_Area01_SelMan" )
      Contact( "Area01".DataIn.PbStop )
   END_RUNG wire#w5
   RUNG wire#powerrail
      Contact( #HMI.B_ConfirmEmptyingShow )
      I_Contact( #ZSI.Door_NormalStop )
      I_Contact( #ZSI.Door_SafeStop )
      I_Contact( #ZSI.Door_Opened )
      Contact( #CIn.Straigtener.Lift_Entry.Rest )
      wire#w6
      Contact( #CIn.Straigtener.Lift_Exit.Rest )
      wire#w7
      Contact( #CIn.JB.CutHead.Rest )
      Contact( #CIn.JB.ClampEntry.Rest )
      Contact( #CIn.JB.ClampExit.Rest )
      Contact( #CIn.JB.Pinchroll_Lift.Rest )
      Coil( #Cnd )
   END_RUNG
   RUNG wire#w6
      Contact( TRUE )
   END_RUNG wire#w7
   RUNG wire#powerrail
      Contact( #TON_Emptying.Q )
      S_SR(operand := #COut.Gen.EmptyingConfirmed, r1 := wire#w8)
   END_RUNG
   RUNG wire#powerrail
      I_Contact( #Cnd )
   END_RUNG wire#w8
   RUNG wire#powerrail
      Contact( #COut.Gen.EmptyingConfirmed )
      Coil( #Warning.EmptyingIsON )
   END_RUNG
   RUNG wire#powerrail
      Contact( #COut.Gen.EmptyingConfirmed )
      Coil( #HMI.B_ConfirmEmptyingStatus )
   END_RUNG
   // the same network as SCL:
   #HMI.B_ConfirmEmptyingShow := (#AreaInterface.Man OR #COut.Gen.EmptyingConfirmed) AND (NOT #Pers.Data.MaterialPresence_StraightenerEntry OR #Pers.Data.MATERIAL_SEPARATION.CutDoneAndConfirmed) AND NOT #Pers.Data.MaterialPresence_StraightenerExit AND (#Sts.EndOfCoil.Idle OR #Sts.EndOfCoil.EndOfSequence);
   #TON_Emptying(IN := (#HMI.B_ConfirmEmptying OR ("MB1_Area01_SelMan" AND "Area01".DataIn.PbStop)) AND #HMI.B_ConfirmEmptyingShow,   // TON
                 PT := T#3s);
   #Cnd := #HMI.B_ConfirmEmptyingShow AND NOT #ZSI.Door_NormalStop AND NOT #ZSI.Door_SafeStop AND NOT #ZSI.Door_Opened AND #CIn.Straigtener.Lift_Entry.Rest AND (#CIn.Straigtener.Lift_Exit.Rest OR TRUE) AND #CIn.JB.CutHead.Rest AND #CIn.JB.ClampEntry.Rest AND #CIn.JB.ClampExit.Rest AND #CIn.JB.Pinchroll_Lift.Rest;
   IF #TON_Emptying.Q THEN
       #COut.Gen.EmptyingConfirmed := TRUE;   // SR flip-flop
   END_IF;
   IF NOT #Cnd THEN #COut.Gen.EmptyingConfirmed := FALSE; END_IF;
   #Warning.EmptyingIsON := #COut.Gen.EmptyingConfirmed;
   #HMI.B_ConfirmEmptyingStatus := #COut.Gen.EmptyingConfirmed;
END_REGION

REGION Network 27: >
END_REGION

REGION Network 28: Material feeding Stop
   RUNG wire#powerrail
      Contact( TRUE )
      Coil( #Sts.EnableCycleStopProgrammed )
   END_RUNG
   RUNG wire#powerrail
      I_Contact( #AreaInterface.StopInPhase )
      I_Contact( #Sts.AlarmsPresence )
      Not()
      wire#w1
      Contact( #AreaInterface.Cycle )
      S_SR(operand := #Ctrl.Stop, r1 := wire#w3)
      R_Coil( #Sts.EnableCycleStopProgrammed )
   END_RUNG
   RUNG wire#powerrail
      Contact( #AreaInterface.StopProgrammed )
      wire#w2
      Contact( #Sts.EnableCycleStopProgrammed )
   END_RUNG wire#w1
   RUNG wire#w2
      Contact( #Ctrl.Stop )
   END_RUNG wire#w1
   RUNG wire#powerrail
      I_Contact( #AreaInterface.Cycle )
      Contact( #Sts.FeedStandstill )
   END_RUNG wire#w3
   // the same network as SCL:
   #Sts.EnableCycleStopProgrammed := TRUE;
   IF (NOT (NOT #AreaInterface.StopInPhase AND NOT #Sts.AlarmsPresence) OR (#AreaInterface.StopProgrammed AND (#Sts.EnableCycleStopProgrammed OR #Ctrl.Stop))) AND #AreaInterface.Cycle THEN
       #Ctrl.Stop := TRUE;   // SR flip-flop
   END_IF;
   IF NOT #AreaInterface.Cycle AND #Sts.FeedStandstill THEN #Ctrl.Stop := FALSE; END_IF;
   IF #Ctrl.Stop THEN #Sts.EnableCycleStopProgrammed := FALSE; END_IF;
END_REGION

REGION Network 29: Material feeding Pause
   RUNG wire#powerrail
      I_Contact( #ZSI.Door_NormalStop )
      I_Contact( #ZSI.Door_SafeStop )
      Not()
      wire#w1
      Coil( #Req )
      S_SR(operand := #Ctrl.Pause, r1 := wire#w2)
   END_RUNG
   RUNG wire#powerrail
      I_Contact( #CIn.Loop.Enable_FWD )
   END_RUNG wire#w1
   RUNG wire#powerrail
      I_Contact( #Req )
      Contact( #Sts.FeedStandstill )
   END_RUNG wire#w2
   RUNG wire#powerrail
      I_Contact( #AreaInterface.Cycle )
   END_RUNG wire#w2
   // the same network as SCL:
   #Req := NOT (NOT #ZSI.Door_NormalStop AND NOT #ZSI.Door_SafeStop) OR NOT #CIn.Loop.Enable_FWD;
   IF #Req THEN
       #Ctrl.Pause := TRUE;   // SR flip-flop
   END_IF;
   IF (NOT #Req AND #Sts.FeedStandstill) OR NOT #AreaInterface.Cycle THEN #Ctrl.Pause := FALSE; END_IF;
END_REGION

REGION Network 30: Material Bkw / Fwd enable
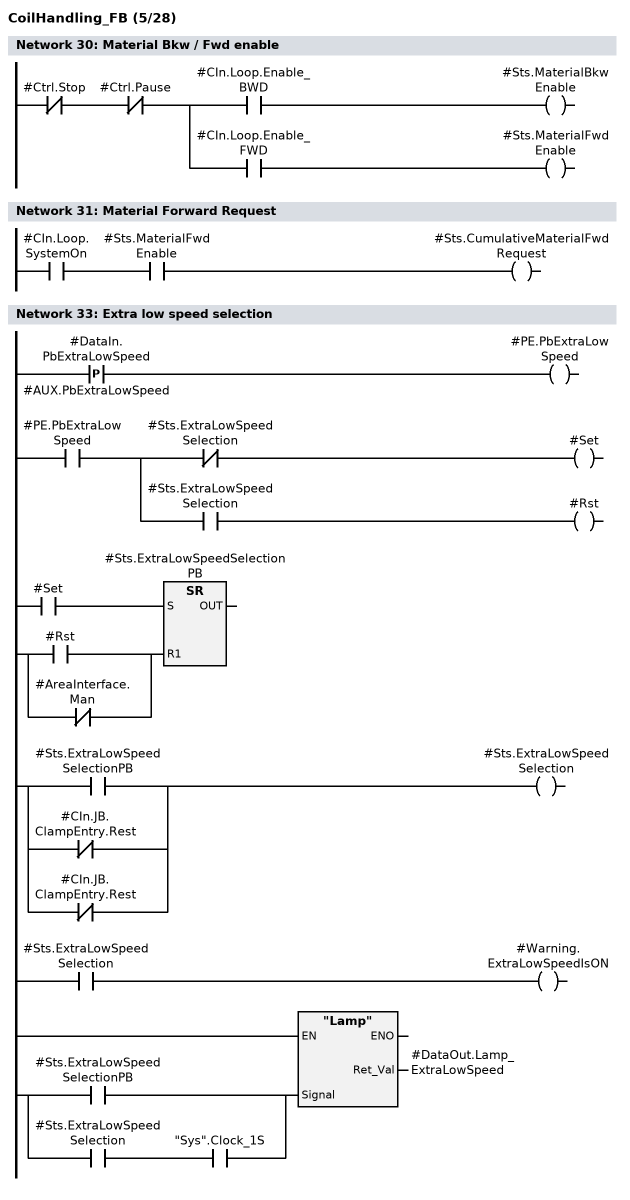
   RUNG wire#powerrail
      I_Contact( #Ctrl.Stop )
      I_Contact( #Ctrl.Pause )
      wire#w1
      Contact( #CIn.Loop.Enable_BWD )
      Coil( #Sts.MaterialBkwEnable )
   END_RUNG
   RUNG wire#w1
      Contact( #CIn.Loop.Enable_FWD )
      Coil( #Sts.MaterialFwdEnable )
   END_RUNG
   // the same network as SCL:
   #_w1 := NOT #Ctrl.Stop AND NOT #Ctrl.Pause;
   #Sts.MaterialBkwEnable := #_w1 AND #CIn.Loop.Enable_BWD;
   #Sts.MaterialFwdEnable := #_w1 AND #CIn.Loop.Enable_FWD;
END_REGION

REGION Network 31: Material Forward Request
   RUNG wire#powerrail
      Contact( #CIn.Loop.SystemOn )
      Contact( #Sts.MaterialFwdEnable )
      Coil( #Sts.CumulativeMaterialFwdRequest )
   END_RUNG
   // the same network as SCL:
   #Sts.CumulativeMaterialFwdRequest := #CIn.Loop.SystemOn AND #Sts.MaterialFwdEnable;
END_REGION

REGION Network 32: <<+>>
END_REGION

REGION Network 33: Extra low speed selection
   RUNG wire#powerrail
      P_Contact(operand := #DataIn.PbExtraLowSpeed, bit := #AUX.PbExtraLowSpeed)
      Coil( #PE.PbExtraLowSpeed )
   END_RUNG
   RUNG wire#powerrail
      Contact( #PE.PbExtraLowSpeed )
      wire#w1
      I_Contact( #Sts.ExtraLowSpeedSelection )
      Coil( #Set )
   END_RUNG
   RUNG wire#w1
      Contact( #Sts.ExtraLowSpeedSelection )
      Coil( #Rst )
   END_RUNG
   RUNG wire#powerrail
      Contact( #Set )
      S_SR(operand := #Sts.ExtraLowSpeedSelectionPB, r1 := wire#w2)
   END_RUNG
   RUNG wire#powerrail
      Contact( #Rst )
   END_RUNG wire#w2
   RUNG wire#powerrail
      I_Contact( #AreaInterface.Man )
   END_RUNG wire#w2
   RUNG wire#powerrail
      Contact( #Sts.ExtraLowSpeedSelectionPB )
      wire#w3
      Coil( #Sts.ExtraLowSpeedSelection )
   END_RUNG
   RUNG wire#powerrail
      I_Contact( #CIn.JB.ClampEntry.Rest )
   END_RUNG wire#w3
   RUNG wire#powerrail
      I_Contact( #CIn.JB.ClampEntry.Rest )
   END_RUNG wire#w3
   RUNG wire#powerrail
      Contact( #Sts.ExtraLowSpeedSelection )
      Coil( #Warning.ExtraLowSpeedIsON )
   END_RUNG
   RUNG wire#powerrail
      "Lamp"(Signal := wire#w4, Ret_Val => #DataOut.Lamp_ExtraLowSpeed)
   END_RUNG
   RUNG wire#powerrail
      Contact( #Sts.ExtraLowSpeedSelectionPB )
   END_RUNG wire#w4
   RUNG wire#powerrail
      Contact( #Sts.ExtraLowSpeedSelection )
      Contact( "Sys".Clock_1S )
   END_RUNG wire#w4
   // the same network as SCL:
   #_w1 := #DataIn.PbExtraLowSpeed AND NOT #AUX.PbExtraLowSpeed;   // rising edge of #DataIn.PbExtraLowSpeed
   #AUX.PbExtraLowSpeed := #DataIn.PbExtraLowSpeed;
   #PE.PbExtraLowSpeed := #_w1;
   #Set := #PE.PbExtraLowSpeed AND NOT #Sts.ExtraLowSpeedSelection;
   #Rst := #PE.PbExtraLowSpeed AND #Sts.ExtraLowSpeedSelection;
   IF #Set THEN
       #Sts.ExtraLowSpeedSelectionPB := TRUE;   // SR flip-flop
   END_IF;
   IF #Rst OR NOT #AreaInterface.Man THEN #Sts.ExtraLowSpeedSelectionPB := FALSE; END_IF;
   #Sts.ExtraLowSpeedSelection := #Sts.ExtraLowSpeedSelectionPB OR NOT #CIn.JB.ClampEntry.Rest OR NOT #CIn.JB.ClampEntry.Rest;
   #Warning.ExtraLowSpeedIsON := #Sts.ExtraLowSpeedSelection;
   #DataOut.Lamp_ExtraLowSpeed := "Lamp"(Signal := #Sts.ExtraLowSpeedSelectionPB OR (#Sts.ExtraLowSpeedSelection AND "Sys".Clock_1S));
END_REGION

REGION Network 34: <<+>>
END_REGION

REGION Network 35: Loop synchro before coil end (using coil diameter)
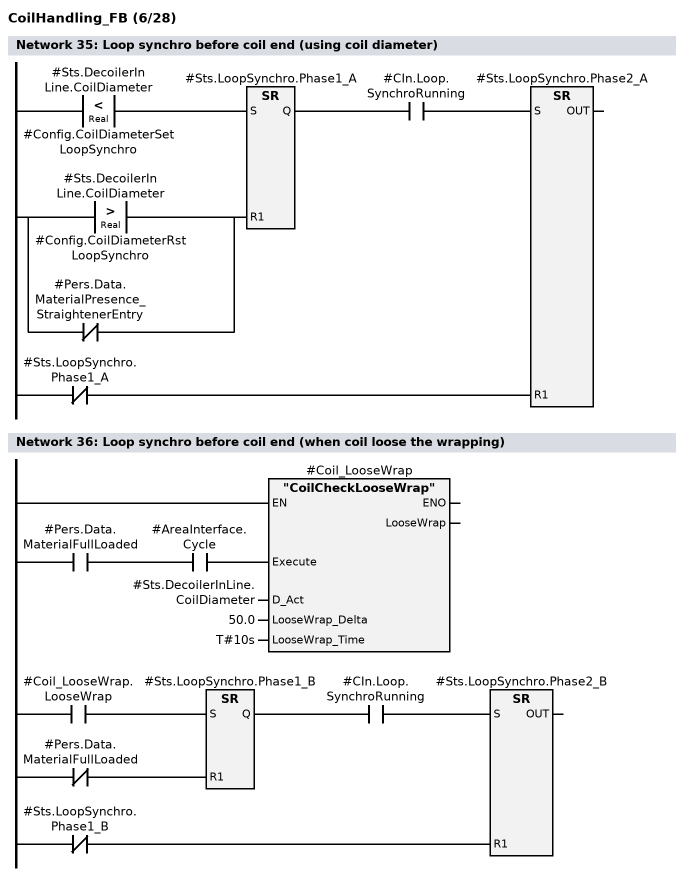
   RUNG wire#powerrail
      { S7_Templates := "SrcType := Real" } LT_Contact(in1 := #Sts.DecoilerInLine.CoilDiameter, in2 := #Config.CoilDiameterSetLoopSynchro)
      S_SR(operand := #Sts.LoopSynchro.Phase1_A, r1 := wire#w1)
      Contact( #CIn.Loop.SynchroRunning )
      S_SR(operand := #Sts.LoopSynchro.Phase2_A, r1 := wire#w2)
   END_RUNG
   RUNG wire#powerrail
      { S7_Templates := "SrcType := Real" } GT_Contact(in1 := #Sts.DecoilerInLine.CoilDiameter, in2 := #Config.CoilDiameterRstLoopSynchro)
   END_RUNG wire#w1
   RUNG wire#powerrail
      I_Contact( #Pers.Data.MaterialPresence_StraightenerEntry )
   END_RUNG wire#w1
   RUNG wire#powerrail
      I_Contact( #Sts.LoopSynchro.Phase1_A )
   END_RUNG wire#w2
   // the same network as SCL:
   IF #Sts.DecoilerInLine.CoilDiameter < #Config.CoilDiameterSetLoopSynchro THEN
       #Sts.LoopSynchro.Phase1_A := TRUE;   // SR flip-flop
   END_IF;
   IF (#Sts.DecoilerInLine.CoilDiameter > #Config.CoilDiameterRstLoopSynchro) OR NOT #Pers.Data.MaterialPresence_StraightenerEntry THEN
       #Sts.LoopSynchro.Phase1_A := FALSE;
   END_IF;
   IF #Sts.LoopSynchro.Phase1_A AND #CIn.Loop.SynchroRunning THEN
       #Sts.LoopSynchro.Phase2_A := TRUE;   // SR flip-flop
   END_IF;
   IF NOT #Sts.LoopSynchro.Phase1_A THEN #Sts.LoopSynchro.Phase2_A := FALSE; END_IF;
END_REGION

REGION Network 36: Loop synchro before coil end (when coil loose the wrapping)
   RUNG wire#powerrail
      #Coil_LooseWrap(Execute := wire#w1, D_Act := #Sts.DecoilerInLine.CoilDiameter, LooseWrap_Delta := 50.0, LooseWrap_Time := T#10s, LooseWrap =>)
   END_RUNG
   RUNG wire#powerrail
      Contact( #Pers.Data.MaterialFullLoaded )
      Contact( #AreaInterface.Cycle )
   END_RUNG wire#w1
   RUNG wire#powerrail
      Contact( #Coil_LooseWrap.LooseWrap )
      S_SR(operand := #Sts.LoopSynchro.Phase1_B, r1 := wire#w2)
      Contact( #CIn.Loop.SynchroRunning )
      S_SR(operand := #Sts.LoopSynchro.Phase2_B, r1 := wire#w3)
   END_RUNG
   RUNG wire#powerrail
      I_Contact( #Pers.Data.MaterialFullLoaded )
   END_RUNG wire#w2
   RUNG wire#powerrail
      I_Contact( #Sts.LoopSynchro.Phase1_B )
   END_RUNG wire#w3
   // the same network as SCL:
   #Coil_LooseWrap(Execute := #Pers.Data.MaterialFullLoaded AND #AreaInterface.Cycle,   // "CoilCheckLooseWrap"
                   D_Act := #Sts.DecoilerInLine.CoilDiameter,
                   LooseWrap_Delta := 50.0,
                   LooseWrap_Time := T#10s);
   IF #Coil_LooseWrap.LooseWrap THEN
       #Sts.LoopSynchro.Phase1_B := TRUE;   // SR flip-flop
   END_IF;
   IF NOT #Pers.Data.MaterialFullLoaded THEN #Sts.LoopSynchro.Phase1_B := FALSE; END_IF;
   IF #Sts.LoopSynchro.Phase1_B AND #CIn.Loop.SynchroRunning THEN
       #Sts.LoopSynchro.Phase2_B := TRUE;   // SR flip-flop
   END_IF;
   IF NOT #Sts.LoopSynchro.Phase1_B THEN #Sts.LoopSynchro.Phase2_B := FALSE; END_IF;
END_REGION

REGION Network 37: <<+>>
END_REGION

REGION Network 38: <<< COIL LOADED MANGMENT >>>
END_REGION

REGION Network 39: Coil loaded mem
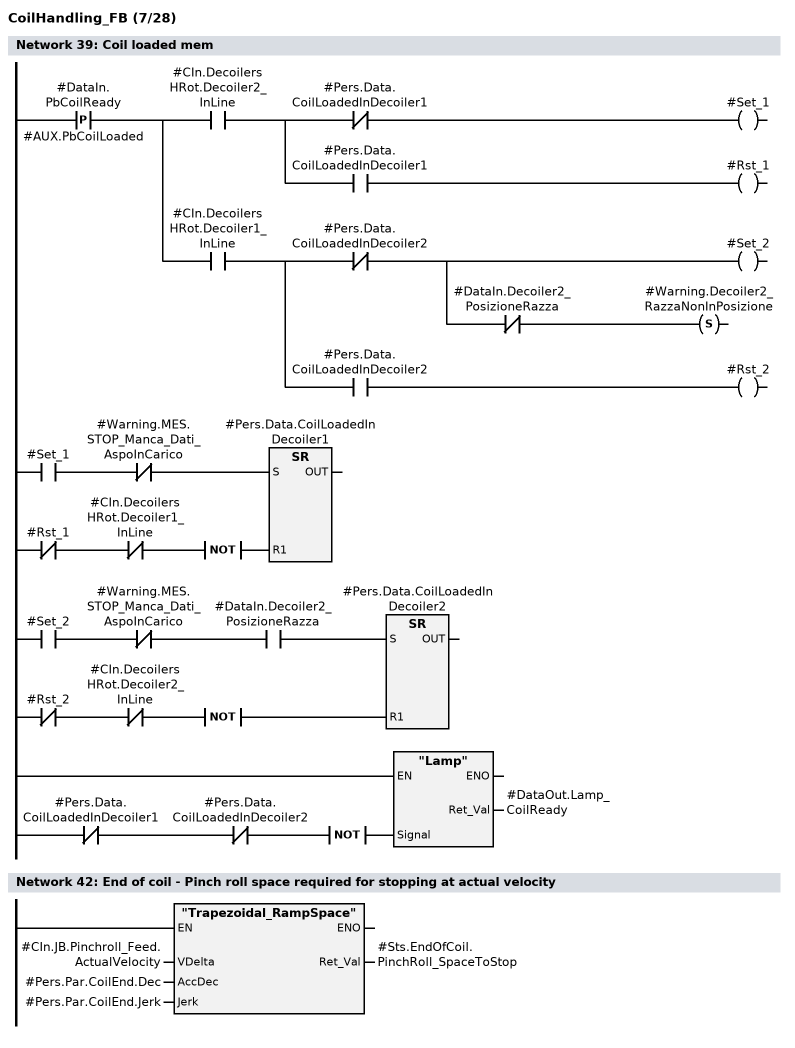
   RUNG wire#powerrail
      P_Contact(operand := #DataIn.PbCoilReady, bit := #AUX.PbCoilLoaded)
      wire#w1
      Contact( #CIn.DecoilersHRot.Decoiler2_InLine )
      wire#w2
      I_Contact( #Pers.Data.CoilLoadedInDecoiler1 )
      Coil( #Set_1 )
   END_RUNG
   RUNG wire#w2
      Contact( #Pers.Data.CoilLoadedInDecoiler1 )
      Coil( #Rst_1 )
   END_RUNG
   RUNG wire#w1
      Contact( #CIn.DecoilersHRot.Decoiler1_InLine )
      wire#w3
      I_Contact( #Pers.Data.CoilLoadedInDecoiler2 )
      wire#w4
      Coil( #Set_2 )
   END_RUNG
   RUNG wire#w4
      I_Contact( #DataIn.Decoiler2_PosizioneRazza )
      S_Coil( #Warning.Decoiler2_RazzaNonInPosizione )
   END_RUNG
   RUNG wire#w3
      Contact( #Pers.Data.CoilLoadedInDecoiler2 )
      Coil( #Rst_2 )
   END_RUNG
   RUNG wire#powerrail
      Contact( #Set_1 )
      I_Contact( #Warning.MES.STOP_Manca_Dati_AspoInCarico )
      S_SR(operand := #Pers.Data.CoilLoadedInDecoiler1, r1 := wire#w5)
   END_RUNG
   RUNG wire#powerrail
      I_Contact( #Rst_1 )
      I_Contact( #CIn.DecoilersHRot.Decoiler1_InLine )
      Not()
   END_RUNG wire#w5
   RUNG wire#powerrail
      Contact( #Set_2 )
      I_Contact( #Warning.MES.STOP_Manca_Dati_AspoInCarico )
      Contact( #DataIn.Decoiler2_PosizioneRazza )
      S_SR(operand := #Pers.Data.CoilLoadedInDecoiler2, r1 := wire#w6)
   END_RUNG
   RUNG wire#powerrail
      I_Contact( #Rst_2 )
      I_Contact( #CIn.DecoilersHRot.Decoiler2_InLine )
      Not()
   END_RUNG wire#w6
   RUNG wire#powerrail
      "Lamp"(Signal := wire#w7, Ret_Val => #DataOut.Lamp_CoilReady)
   END_RUNG
   RUNG wire#powerrail
      I_Contact( #Pers.Data.CoilLoadedInDecoiler1 )
      I_Contact( #Pers.Data.CoilLoadedInDecoiler2 )
      Not()
   END_RUNG wire#w7
   // the same network as SCL:
   #_w1 := #DataIn.PbCoilReady AND NOT #AUX.PbCoilLoaded;   // rising edge of #DataIn.PbCoilReady
   #AUX.PbCoilLoaded := #DataIn.PbCoilReady;
   #_w2 := #_w1 AND #CIn.DecoilersHRot.Decoiler2_InLine;
   #Set_1 := #_w2 AND NOT #Pers.Data.CoilLoadedInDecoiler1;
   #Rst_1 := #_w2 AND #Pers.Data.CoilLoadedInDecoiler1;
   #_w3 := #_w1 AND #CIn.DecoilersHRot.Decoiler1_InLine;
   #Set_2 := #_w3 AND NOT #Pers.Data.CoilLoadedInDecoiler2;
   IF #Set_2 AND NOT #DataIn.Decoiler2_PosizioneRazza THEN
       #Warning.Decoiler2_RazzaNonInPosizione := TRUE;
   END_IF;
   #Rst_2 := #_w3 AND #Pers.Data.CoilLoadedInDecoiler2;
   IF #Set_1 AND NOT #Warning.MES.STOP_Manca_Dati_AspoInCarico THEN
       #Pers.Data.CoilLoadedInDecoiler1 := TRUE;   // SR flip-flop
   END_IF;
   IF NOT (NOT #Rst_1 AND NOT #CIn.DecoilersHRot.Decoiler1_InLine) THEN
       #Pers.Data.CoilLoadedInDecoiler1 := FALSE;
   END_IF;
   IF #Set_2 AND NOT #Warning.MES.STOP_Manca_Dati_AspoInCarico AND #DataIn.Decoiler2_PosizioneRazza THEN
       #Pers.Data.CoilLoadedInDecoiler2 := TRUE;   // SR flip-flop
   END_IF;
   IF NOT (NOT #Rst_2 AND NOT #CIn.DecoilersHRot.Decoiler2_InLine) THEN
       #Pers.Data.CoilLoadedInDecoiler2 := FALSE;
   END_IF;
   #DataOut.Lamp_CoilReady := "Lamp"(Signal := NOT (NOT #Pers.Data.CoilLoadedInDecoiler1 AND NOT #Pers.Data.CoilLoadedInDecoiler2));
END_REGION

REGION Network 40: <<+>>
END_REGION

REGION Network 41: <<< END OF COIL SEQUENCE >>>
END_REGION

REGION Network 42: End of coil - Pinch roll space required for stopping at actual velocity
   RUNG wire#powerrail
      "Trapezoidal_RampSpace"(VDelta := #CIn.JB.Pinchroll_Feed.ActualVelocity, AccDec := #Pers.Par.CoilEnd.Dec, Jerk := #Pers.Par.CoilEnd.Jerk, Ret_Val => #Sts.EndOfCoil.PinchRoll_SpaceToStop)
   END_RUNG
   // the same network as SCL:
   #Sts.EndOfCoil.PinchRoll_SpaceToStop := "Trapezoidal_RampSpace"(VDelta := #CIn.JB.Pinchroll_Feed.ActualVelocity,
                           AccDec := #Pers.Par.CoilEnd.Dec,
                           Jerk := #Pers.Par.CoilEnd.Jerk);
END_REGION

REGION Network 43: End of coil - Save positon
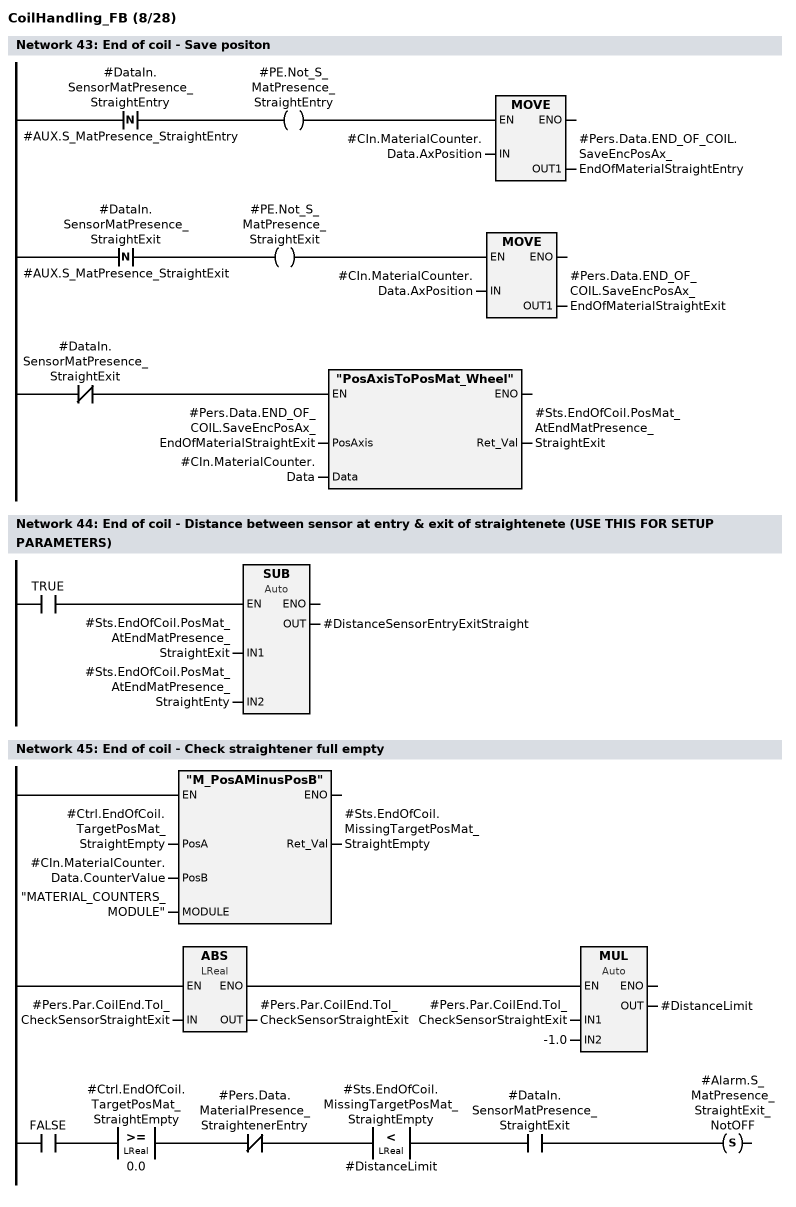
   RUNG wire#powerrail
      N_Contact(operand := #DataIn.SensorMatPresence_StraightEntry, bit := #AUX.S_MatPresence_StraightEntry)
      Coil( #PE.Not_S_MatPresence_StraightEntry )
      Move(in := #CIn.MaterialCounter.Data.AxPosition, out1 => #Pers.Data.END_OF_COIL.SaveEncPosAx_EndOfMaterialStraightEntry)
   END_RUNG
   RUNG wire#powerrail
      N_Contact(operand := #DataIn.SensorMatPresence_StraightExit, bit := #AUX.S_MatPresence_StraightExit)
      Coil( #PE.Not_S_MatPresence_StraightExit )
      Move(in := #CIn.MaterialCounter.Data.AxPosition, out1 => #Pers.Data.END_OF_COIL.SaveEncPosAx_EndOfMaterialStraightExit)
   END_RUNG
   RUNG wire#powerrail
      I_Contact( #DataIn.SensorMatPresence_StraightExit )
      "PosAxisToPosMat_Wheel"(PosAxis := #Pers.Data.END_OF_COIL.SaveEncPosAx_EndOfMaterialStraightExit, Data := #CIn.MaterialCounter.Data, Ret_Val => #Sts.EndOfCoil.PosMat_AtEndMatPresence_StraightExit)
   END_RUNG
   // the same network as SCL:
   #_w1 := NOT #DataIn.SensorMatPresence_StraightEntry AND #AUX.S_MatPresence_StraightEntry;   // falling edge of #DataIn.SensorMatPresence_StraightEntry
   #AUX.S_MatPresence_StraightEntry := #DataIn.SensorMatPresence_StraightEntry;
   #PE.Not_S_MatPresence_StraightEntry := #_w1;
   IF #_w1 THEN
       #Pers.Data.END_OF_COIL.SaveEncPosAx_EndOfMaterialStraightEntry := #CIn.MaterialCounter.Data.AxPosition;
   END_IF;
   #_w2 := NOT #DataIn.SensorMatPresence_StraightExit AND #AUX.S_MatPresence_StraightExit;   // falling edge of #DataIn.SensorMatPresence_StraightExit
   #AUX.S_MatPresence_StraightExit := #DataIn.SensorMatPresence_StraightExit;
   #PE.Not_S_MatPresence_StraightExit := #_w2;
   IF #_w2 THEN
       #Pers.Data.END_OF_COIL.SaveEncPosAx_EndOfMaterialStraightExit := #CIn.MaterialCounter.Data.AxPosition;
   END_IF;
   IF NOT #DataIn.SensorMatPresence_StraightExit THEN
       #Sts.EndOfCoil.PosMat_AtEndMatPresence_StraightExit := "PosAxisToPosMat_Wheel"(PosAxis := #Pers.Data.END_OF_COIL.SaveEncPosAx_EndOfMaterialStraightExit,
                               Data := #CIn.MaterialCounter.Data);
   END_IF;
END_REGION

REGION Network 44: End of coil - Distance between sensor at entry & exit of straightenete (USE THIS FOR SETUP PARAMETERS)
   RUNG wire#powerrail
      Contact( TRUE )
      Sub(in1 := #Sts.EndOfCoil.PosMat_AtEndMatPresence_StraightExit, in2 := #Sts.EndOfCoil.PosMat_AtEndMatPresence_StraightEnty, out => #DistanceSensorEntryExitStraight)
   END_RUNG
   // the same network as SCL:
   IF TRUE THEN
       #DistanceSensorEntryExitStraight := #Sts.EndOfCoil.PosMat_AtEndMatPresence_StraightExit - #Sts.EndOfCoil.PosMat_AtEndMatPresence_StraightEnty;
   END_IF;
END_REGION

REGION Network 45: End of coil - Check straightener full empty
   RUNG wire#powerrail
      "M_PosAMinusPosB"(PosA := #Ctrl.EndOfCoil.TargetPosMat_StraightEmpty, PosB := #CIn.MaterialCounter.Data.CounterValue, MODULE := "MATERIAL_COUNTERS_MODULE", Ret_Val => #Sts.EndOfCoil.MissingTargetPosMat_StraightEmpty)
   END_RUNG
   RUNG wire#powerrail
      { S7_Templates := "SrcType := LReal" } Abs(in := #Pers.Par.CoilEnd.Tol_CheckSensorStraightExit, out => #Pers.Par.CoilEnd.Tol_CheckSensorStraightExit)
      Mul(in1 := #Pers.Par.CoilEnd.Tol_CheckSensorStraightExit, in2 := -1.0, out => #DistanceLimit)
   END_RUNG
   RUNG wire#powerrail
      Contact( FALSE )
      { S7_Templates := "SrcType := LReal" } GE_Contact(in1 := #Ctrl.EndOfCoil.TargetPosMat_StraightEmpty, in2 := 0.0)
      I_Contact( #Pers.Data.MaterialPresence_StraightenerEntry )
      { S7_Templates := "SrcType := LReal" } LT_Contact(in1 := #Sts.EndOfCoil.MissingTargetPosMat_StraightEmpty, in2 := #DistanceLimit)
      Contact( #DataIn.SensorMatPresence_StraightExit )
      S_Coil( #Alarm.S_MatPresence_StraightExit_NotOFF )
   END_RUNG
   // the same network as SCL:
   #Sts.EndOfCoil.MissingTargetPosMat_StraightEmpty := "M_PosAMinusPosB"(PosA := #Ctrl.EndOfCoil.TargetPosMat_StraightEmpty,
                           PosB := #CIn.MaterialCounter.Data.CounterValue,
                           MODULE := "MATERIAL_COUNTERS_MODULE");
   #Pers.Par.CoilEnd.Tol_CheckSensorStraightExit := ABS(#Pers.Par.CoilEnd.Tol_CheckSensorStraightExit);
   #DistanceLimit := #Pers.Par.CoilEnd.Tol_CheckSensorStraightExit * (-1.0);
   IF FALSE AND (#Ctrl.EndOfCoil.TargetPosMat_StraightEmpty >= 0.0) AND NOT #Pers.Data.MaterialPresence_StraightenerEntry AND (#Sts.EndOfCoil.MissingTargetPosMat_StraightEmpty < #DistanceLimit) AND #DataIn.SensorMatPresence_StraightExit THEN
       #Alarm.S_MatPresence_StraightExit_NotOFF := TRUE;
   END_IF;
END_REGION

REGION Network 46: End of coil - Positioning to cut-off execution target
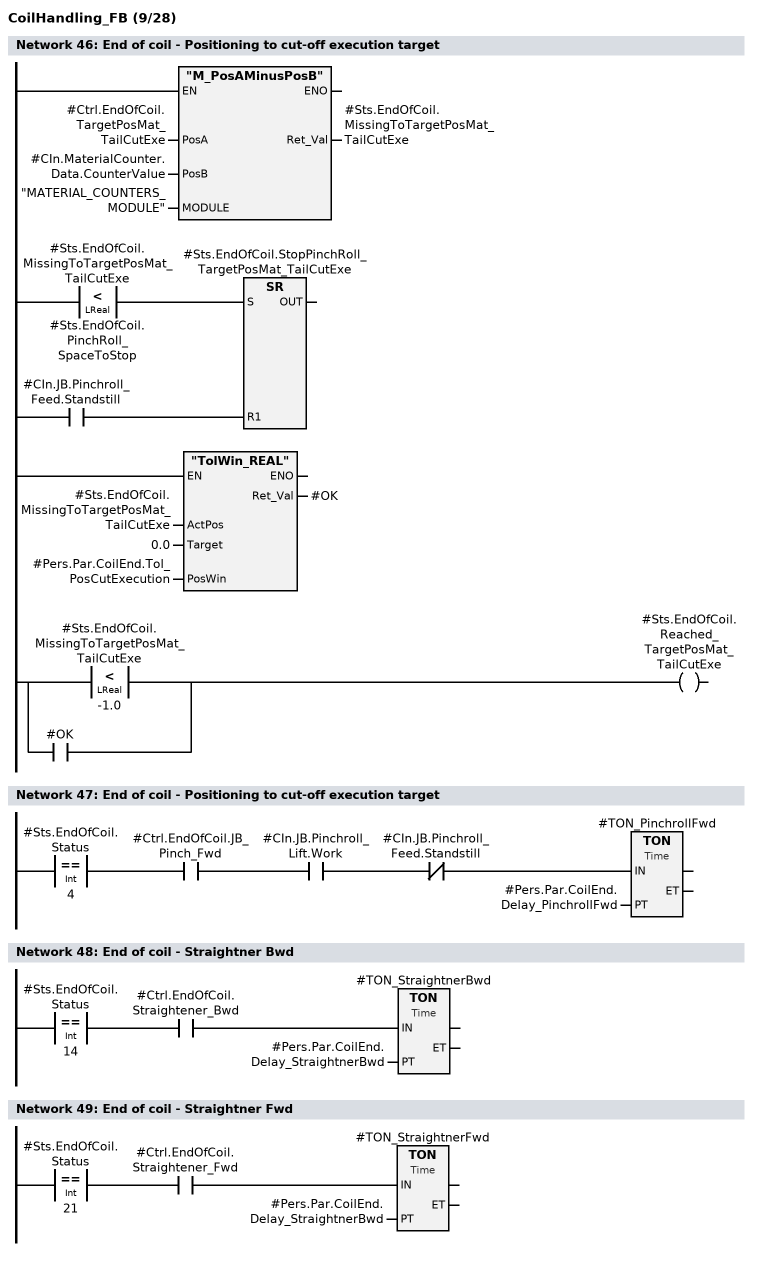
   RUNG wire#powerrail
      "M_PosAMinusPosB"(PosA := #Ctrl.EndOfCoil.TargetPosMat_TailCutExe, PosB := #CIn.MaterialCounter.Data.CounterValue, MODULE := "MATERIAL_COUNTERS_MODULE", Ret_Val => #Sts.EndOfCoil.MissingToTargetPosMat_TailCutExe)
   END_RUNG
   RUNG wire#powerrail
      { S7_Templates := "SrcType := LReal" } LT_Contact(in1 := #Sts.EndOfCoil.MissingToTargetPosMat_TailCutExe, in2 := #Sts.EndOfCoil.PinchRoll_SpaceToStop)
      S_SR(operand := #Sts.EndOfCoil.StopPinchRoll_TargetPosMat_TailCutExe, r1 := wire#w1)
   END_RUNG
   RUNG wire#powerrail
      Contact( #CIn.JB.Pinchroll_Feed.Standstill )
   END_RUNG wire#w1
   RUNG wire#powerrail
      "TolWin_REAL"(ActPos := #Sts.EndOfCoil.MissingToTargetPosMat_TailCutExe, Target := 0.0, PosWin := #Pers.Par.CoilEnd.Tol_PosCutExecution, Ret_Val => #OK)
   END_RUNG
   RUNG wire#powerrail
      { S7_Templates := "SrcType := LReal" } LT_Contact(in1 := #Sts.EndOfCoil.MissingToTargetPosMat_TailCutExe, in2 := -1.0)
      wire#w2
      Coil( #Sts.EndOfCoil.Reached_TargetPosMat_TailCutExe )
   END_RUNG
   RUNG wire#powerrail
      Contact( #OK )
   END_RUNG wire#w2
   // the same network as SCL:
   #Sts.EndOfCoil.MissingToTargetPosMat_TailCutExe := "M_PosAMinusPosB"(PosA := #Ctrl.EndOfCoil.TargetPosMat_TailCutExe,
                           PosB := #CIn.MaterialCounter.Data.CounterValue,
                           MODULE := "MATERIAL_COUNTERS_MODULE");
   IF #Sts.EndOfCoil.MissingToTargetPosMat_TailCutExe < #Sts.EndOfCoil.PinchRoll_SpaceToStop THEN
       #Sts.EndOfCoil.StopPinchRoll_TargetPosMat_TailCutExe := TRUE;   // SR flip-flop
   END_IF;
   IF #CIn.JB.Pinchroll_Feed.Standstill THEN
       #Sts.EndOfCoil.StopPinchRoll_TargetPosMat_TailCutExe := FALSE;
   END_IF;
   #OK := "TolWin_REAL"(ActPos := #Sts.EndOfCoil.MissingToTargetPosMat_TailCutExe,
                        Target := 0.0,
                        PosWin := #Pers.Par.CoilEnd.Tol_PosCutExecution);
   #Sts.EndOfCoil.Reached_TargetPosMat_TailCutExe := (#Sts.EndOfCoil.MissingToTargetPosMat_TailCutExe < (-1.0)) OR #OK;
END_REGION

REGION Network 47: End of coil - Positioning to cut-off execution target
   RUNG wire#powerrail
      { S7_Templates := "SrcType := Int" } EQ_Contact(in1 := #Sts.EndOfCoil.Status, in2 := 4)
      Contact( #Ctrl.EndOfCoil.JB_Pinch_Fwd )
      Contact( #CIn.JB.Pinchroll_Lift.Work )
      I_Contact( #CIn.JB.Pinchroll_Feed.Standstill )
      { S7_Templates := "time_type := Time" } #TON_PinchrollFwd.TON(pt := #Pers.Par.CoilEnd.Delay_PinchrollFwd, et =>)
   END_RUNG
   // the same network as SCL:
   #TON_PinchrollFwd(IN := (#Sts.EndOfCoil.Status = 4) AND #Ctrl.EndOfCoil.JB_Pinch_Fwd AND #CIn.JB.Pinchroll_Lift.Work AND NOT #CIn.JB.Pinchroll_Feed.Standstill,   // TON
                     PT := #Pers.Par.CoilEnd.Delay_PinchrollFwd);
END_REGION

REGION Network 48: End of coil - Straightner Bwd
   RUNG wire#powerrail
      { S7_Templates := "SrcType := Int" } EQ_Contact(in1 := #Sts.EndOfCoil.Status, in2 := 14)
      Contact( #Ctrl.EndOfCoil.Straightener_Bwd )
      { S7_Templates := "time_type := Time" } #TON_StraightnerBwd.TON(pt := #Pers.Par.CoilEnd.Delay_StraightnerBwd, et =>)
   END_RUNG
   // the same network as SCL:
   #TON_StraightnerBwd(IN := (#Sts.EndOfCoil.Status = 14) AND #Ctrl.EndOfCoil.Straightener_Bwd,   // TON
                       PT := #Pers.Par.CoilEnd.Delay_StraightnerBwd);
END_REGION

REGION Network 49: End of coil - Straightner Fwd
   RUNG wire#powerrail
      { S7_Templates := "SrcType := Int" } EQ_Contact(in1 := #Sts.EndOfCoil.Status, in2 := 21)
      Contact( #Ctrl.EndOfCoil.Straightener_Fwd )
      { S7_Templates := "time_type := Time" } #TON_StraightnerFwd.TON(pt := #Pers.Par.CoilEnd.Delay_StraightnerBwd, et =>)
   END_RUNG
   // the same network as SCL:
   #TON_StraightnerFwd(IN := (#Sts.EndOfCoil.Status = 21) AND #Ctrl.EndOfCoil.Straightener_Fwd,   // TON
                       PT := #Pers.Par.CoilEnd.Delay_StraightnerBwd);
END_REGION

REGION Network 50: End of coil - Positioning to junction execution target
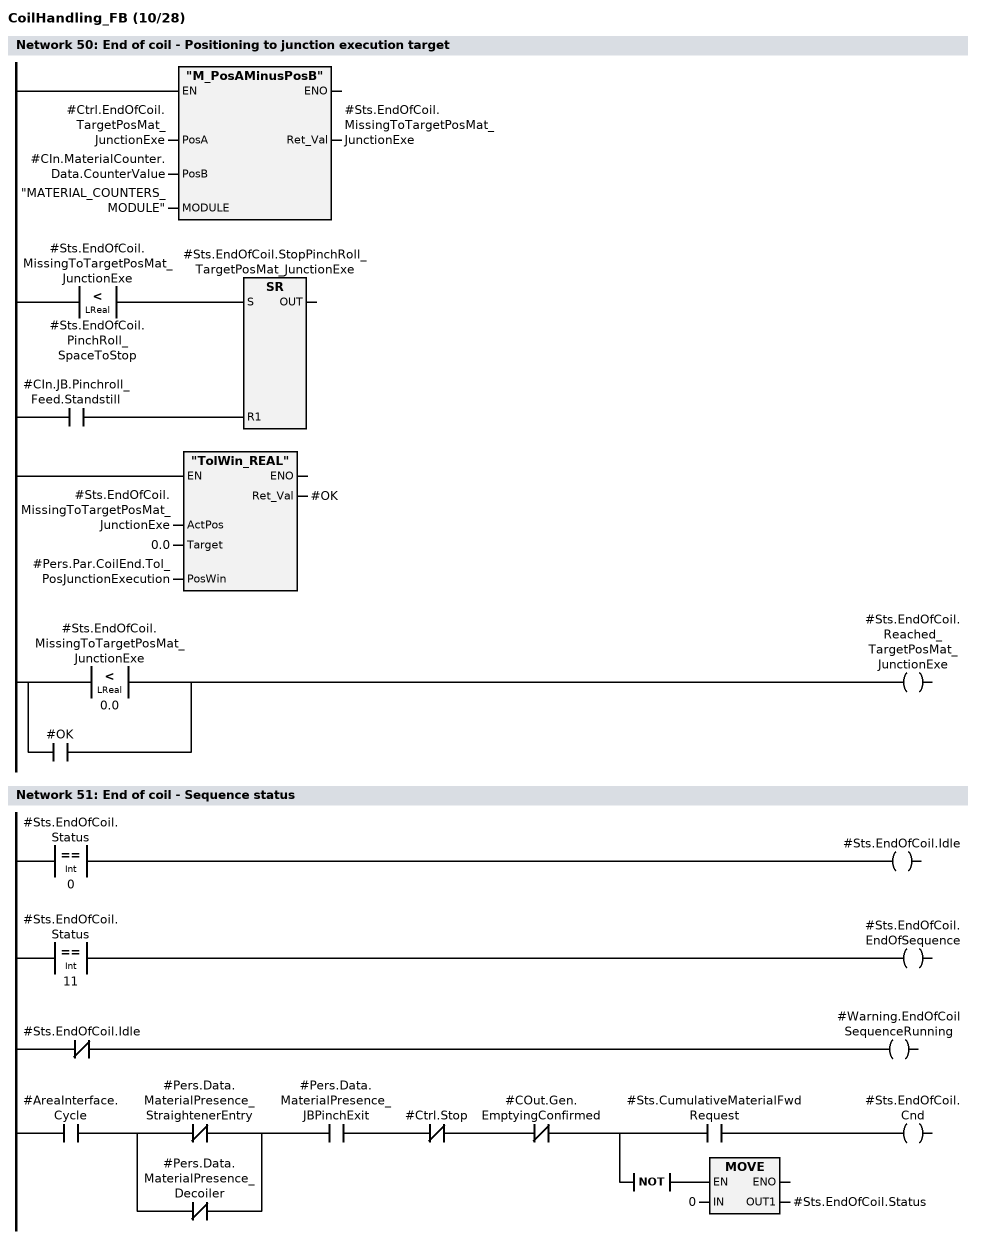
   RUNG wire#powerrail
      "M_PosAMinusPosB"(PosA := #Ctrl.EndOfCoil.TargetPosMat_JunctionExe, PosB := #CIn.MaterialCounter.Data.CounterValue, MODULE := "MATERIAL_COUNTERS_MODULE", Ret_Val => #Sts.EndOfCoil.MissingToTargetPosMat_JunctionExe)
   END_RUNG
   RUNG wire#powerrail
      { S7_Templates := "SrcType := LReal" } LT_Contact(in1 := #Sts.EndOfCoil.MissingToTargetPosMat_JunctionExe, in2 := #Sts.EndOfCoil.PinchRoll_SpaceToStop)
      S_SR(operand := #Sts.EndOfCoil.StopPinchRoll_TargetPosMat_JunctionExe, r1 := wire#w1)
   END_RUNG
   RUNG wire#powerrail
      Contact( #CIn.JB.Pinchroll_Feed.Standstill )
   END_RUNG wire#w1
   RUNG wire#powerrail
      "TolWin_REAL"(ActPos := #Sts.EndOfCoil.MissingToTargetPosMat_JunctionExe, Target := 0.0, PosWin := #Pers.Par.CoilEnd.Tol_PosJunctionExecution, Ret_Val => #OK)
   END_RUNG
   RUNG wire#powerrail
      { S7_Templates := "SrcType := LReal" } LT_Contact(in1 := #Sts.EndOfCoil.MissingToTargetPosMat_JunctionExe, in2 := 0.0)
      wire#w2
      Coil( #Sts.EndOfCoil.Reached_TargetPosMat_JunctionExe )
   END_RUNG
   RUNG wire#powerrail
      Contact( #OK )
   END_RUNG wire#w2
   // the same network as SCL:
   #Sts.EndOfCoil.MissingToTargetPosMat_JunctionExe := "M_PosAMinusPosB"(PosA := #Ctrl.EndOfCoil.TargetPosMat_JunctionExe,
                           PosB := #CIn.MaterialCounter.Data.CounterValue,
                           MODULE := "MATERIAL_COUNTERS_MODULE");
   IF #Sts.EndOfCoil.MissingToTargetPosMat_JunctionExe < #Sts.EndOfCoil.PinchRoll_SpaceToStop THEN
       #Sts.EndOfCoil.StopPinchRoll_TargetPosMat_JunctionExe := TRUE;   // SR flip-flop
   END_IF;
   IF #CIn.JB.Pinchroll_Feed.Standstill THEN
       #Sts.EndOfCoil.StopPinchRoll_TargetPosMat_JunctionExe := FALSE;
   END_IF;
   #OK := "TolWin_REAL"(ActPos := #Sts.EndOfCoil.MissingToTargetPosMat_JunctionExe,
                        Target := 0.0,
                        PosWin := #Pers.Par.CoilEnd.Tol_PosJunctionExecution);
   #Sts.EndOfCoil.Reached_TargetPosMat_JunctionExe := (#Sts.EndOfCoil.MissingToTargetPosMat_JunctionExe < 0.0) OR #OK;
END_REGION

REGION Network 51: End of coil - Sequence status
   RUNG wire#powerrail
      { S7_Templates := "SrcType := Int" } EQ_Contact(in1 := #Sts.EndOfCoil.Status, in2 := 0)
      Coil( #Sts.EndOfCoil.Idle )
   END_RUNG
   RUNG wire#powerrail
      { S7_Templates := "SrcType := Int" } EQ_Contact(in1 := #Sts.EndOfCoil.Status, in2 := 11)
      Coil( #Sts.EndOfCoil.EndOfSequence )
   END_RUNG
   RUNG wire#powerrail
      I_Contact( #Sts.EndOfCoil.Idle )
      Coil( #Warning.EndOfCoilSequenceRunning )
   END_RUNG
   RUNG wire#powerrail
      Contact( #AreaInterface.Cycle )
      wire#w1
      I_Contact( #Pers.Data.MaterialPresence_StraightenerEntry )
      wire#w2
      Contact( #Pers.Data.MaterialPresence_JBPinchExit )
      I_Contact( #Ctrl.Stop )
      I_Contact( #COut.Gen.EmptyingConfirmed )
      wire#w3
      Contact( #Sts.CumulativeMaterialFwdRequest )
      Coil( #Sts.EndOfCoil.Cnd )
   END_RUNG
   RUNG wire#w1
      I_Contact( #Pers.Data.MaterialPresence_Decoiler )
   END_RUNG wire#w2
   RUNG wire#w3
      Not()
      Move(in := 0, out1 => #Sts.EndOfCoil.Status)
   END_RUNG
   // the same network as SCL:
   #Sts.EndOfCoil.Idle := #Sts.EndOfCoil.Status = 0;
   #Sts.EndOfCoil.EndOfSequence := #Sts.EndOfCoil.Status = 11;
   #Warning.EndOfCoilSequenceRunning := NOT #Sts.EndOfCoil.Idle;
   #_w1 := #AreaInterface.Cycle AND (NOT #Pers.Data.MaterialPresence_StraightenerEntry OR NOT #Pers.Data.MaterialPresence_Decoiler) AND #Pers.Data.MaterialPresence_JBPinchExit AND NOT #Ctrl.Stop AND NOT #COut.Gen.EmptyingConfirmed;
   #Sts.EndOfCoil.Cnd := #_w1 AND #Sts.CumulativeMaterialFwdRequest;
   IF NOT #_w1 THEN #Sts.EndOfCoil.Status := 0; END_IF;
END_REGION

REGION Network 52: End of coil - Target
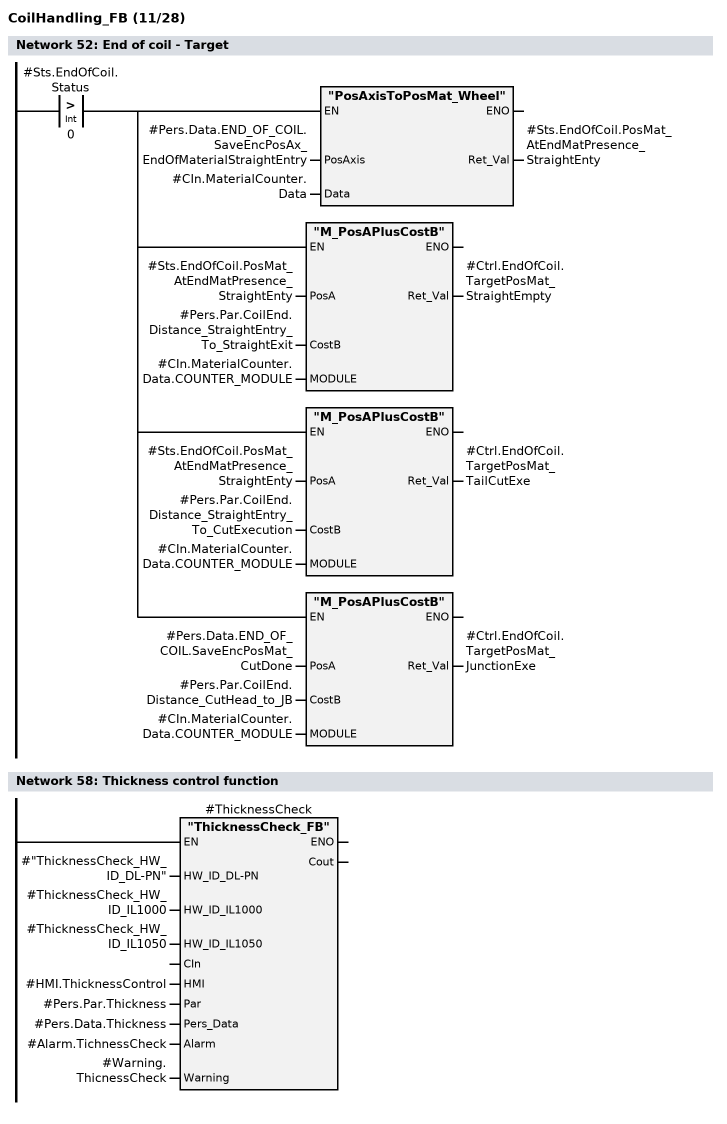
   RUNG wire#powerrail
      { S7_Templates := "SrcType := Int" } GT_Contact(in1 := #Sts.EndOfCoil.Status, in2 := 0)
      wire#w1
      "PosAxisToPosMat_Wheel"(PosAxis := #Pers.Data.END_OF_COIL.SaveEncPosAx_EndOfMaterialStraightEntry, Data := #CIn.MaterialCounter.Data, Ret_Val => #Sts.EndOfCoil.PosMat_AtEndMatPresence_StraightEnty)
   END_RUNG
   RUNG wire#w1
      "M_PosAPlusCostB"(PosA := #Sts.EndOfCoil.PosMat_AtEndMatPresence_StraightEnty, CostB := #Pers.Par.CoilEnd.Distance_StraightEntry_To_StraightExit, MODULE := #CIn.MaterialCounter.Data.COUNTER_MODULE, Ret_Val => #Ctrl.EndOfCoil.TargetPosMat_StraightEmpty)
   END_RUNG
   RUNG wire#w1
      "M_PosAPlusCostB"(PosA := #Sts.EndOfCoil.PosMat_AtEndMatPresence_StraightEnty, CostB := #Pers.Par.CoilEnd.Distance_StraightEntry_To_CutExecution, MODULE := #CIn.MaterialCounter.Data.COUNTER_MODULE, Ret_Val => #Ctrl.EndOfCoil.TargetPosMat_TailCutExe)
   END_RUNG
   RUNG wire#w1
      "M_PosAPlusCostB"(PosA := #Pers.Data.END_OF_COIL.SaveEncPosMat_CutDone, CostB := #Pers.Par.CoilEnd.Distance_CutHead_to_JB, MODULE := #CIn.MaterialCounter.Data.COUNTER_MODULE, Ret_Val => #Ctrl.EndOfCoil.TargetPosMat_JunctionExe)
   END_RUNG
   // the same network as SCL:
   IF #Sts.EndOfCoil.Status > 0 THEN
       #Sts.EndOfCoil.PosMat_AtEndMatPresence_StraightEnty := "PosAxisToPosMat_Wheel"(PosAxis := #Pers.Data.END_OF_COIL.SaveEncPosAx_EndOfMaterialStraightEntry,
                               Data := #CIn.MaterialCounter.Data);
       #Ctrl.EndOfCoil.TargetPosMat_StraightEmpty := "M_PosAPlusCostB"(PosA := #Sts.EndOfCoil.PosMat_AtEndMatPresence_StraightEnty,
                               CostB := #Pers.Par.CoilEnd.Distance_StraightEntry_To_StraightExit,
                               MODULE := #CIn.MaterialCounter.Data.COUNTER_MODULE);
       #Ctrl.EndOfCoil.TargetPosMat_TailCutExe := "M_PosAPlusCostB"(PosA := #Sts.EndOfCoil.PosMat_AtEndMatPresence_StraightEnty,
                               CostB := #Pers.Par.CoilEnd.Distance_StraightEntry_To_CutExecution,
                               MODULE := #CIn.MaterialCounter.Data.COUNTER_MODULE);
       #Ctrl.EndOfCoil.TargetPosMat_JunctionExe := "M_PosAPlusCostB"(PosA := #Pers.Data.END_OF_COIL.SaveEncPosMat_CutDone,
                               CostB := #Pers.Par.CoilEnd.Distance_CutHead_to_JB,
                               MODULE := #CIn.MaterialCounter.Data.COUNTER_MODULE);
   END_IF;
END_REGION

REGION Network 53 (SCL): End of coil - Sequence


   CASE #Sts.EndOfCoil.Status OF


           //#######################################################################################################
           // Status = 0 - Wait end of coil for starting sequence
           //#######################################################################################################
           //
       0:
           // Reset controls
           #Ctrl.EndOfCoil.StraightRollEntry_Open := FALSE;
           #Ctrl.EndOfCoil.StraightRollEntry_Close := FALSE;
           #Ctrl.EndOfCoil.Straightener_Bwd := FALSE;
           #Ctrl.EndOfCoil.Straightener_Fwd := FALSE;
           #Ctrl.EndOfCoil.JB_Pinch_Close := FALSE;
           #Ctrl.EndOfCoil.JB_Pinch_Fwd := FALSE;
           #Ctrl.EndOfCoil.JB_Cut_Rest := FALSE;
           #Ctrl.EndOfCoil.JB_Cut_Work := FALSE;
           #Ctrl.EndOfCoil.JB_Welder_Open := FALSE;
           #Ctrl.EndOfCoil.TargetPosMat_StraightEmpty := -1.0;
           #Ctrl.EndOfCoil.TargetPosMat_TailCutExe := -1.0;
           #Ctrl.EndOfCoil.TargetPosMat_JunctionExe := -1.0;
           #Ctrl.EndOfCoil.ChangeCoilExe := FALSE;
           #Ctrl.EndOfCoil.Decoiler_Fwd := FALSE;

           // Start when conditons met
           IF #Sts.EndOfCoil.Cnd THEN
               #Sts.EndOfCoil.Status += 1;

           ELSIF NOT #Pers.Data.MaterialPresence_StraightenerEntry THEN
               // Reset memories
               #Pers.Data.END_OF_COIL.Tail_ReachCutPosition := FALSE;
               #Pers.Data.END_OF_COIL.Tail_CutDone := FALSE;
               #Pers.Data.END_OF_COIL.Tail_ReachJunctionPos := FALSE;

           END_IF;



           //#######################################################################################################
           // Status = 1 - Close roll of pinch roll + Close rolls of straightener + Open JB clamps
           //#######################################################################################################
           //
       1:

           #Ctrl.EndOfCoil.JB_Pinch_Close := NOT #CIn.JB.Pinchroll_Lift.Work;

           #Ctrl.EndOfCoil.StraightRollEntry_Close := NOT #CIn.Straigtener.Lift_Entry.Work AND #StraightRollEntry_Used;
           #Ctrl.EndOfCoil.StraightRollExit_Close := NOT #CIn.Straigtener.Lift_Exit.Work AND #StraightRollExit_Used;

           #Ctrl.EndOfCoil.JB_Welder_Open := NOT #CIn.JB.ClampEntry.Rest OR NOT #CIn.JB.ClampExit.Rest ;
           #Ctrl.EndOfCoil.JB_Cut_Rest := NOT #CIn.JB.CutHead.Rest;


           IF NOT #Ctrl.EndOfCoil.JB_Pinch_Close
               AND
               NOT #Ctrl.EndOfCoil.StraightRollEntry_Close
               AND
               NOT #Ctrl.EndOfCoil.StraightRollExit_Close
               AND
               NOT #Ctrl.EndOfCoil.JB_Welder_Open
               AND
               NOT #Ctrl.EndOfCoil.JB_Cut_Rest
           THEN

               IF #Pers.Par.CoilEnd.EnableCoilTailSequence THEN
                   // #Sts.EndOfCoil.Status += 1;
                   #Sts.EndOfCoil.Status := 20;
               ELSE
                   #Sts.EndOfCoil.Status := 10; // jump to end of sequence 
               END_IF;
           END_IF;


           //#######################################################################################################
           // Status = 2 - Fwd Pinchroll + Straightener for material extraction from straightener
           //#######################################################################################################    

       2:

           #Ctrl.EndOfCoil.JB_Pinch_Fwd := #Pers.Data.MaterialPresence_StraightenerExit;
           #Ctrl.EndOfCoil.Straightener_Fwd := #Ctrl.EndOfCoil.JB_Pinch_Fwd;

           IF #Alarm.S_MatPresence_StraightExit_NotOFF
           THEN
               #Sts.EndOfCoil.Status := 99;

           ELSIF NOT #Ctrl.EndOfCoil.JB_Pinch_Fwd
           THEN
               #Sts.EndOfCoil.Status += 1;
           END_IF;


           //#######################################################################################################
           // Status = 3 - Open rolls of straightener
           //#######################################################################################################    
       3:

           #Ctrl.EndOfCoil.StraightRollEntry_Open := NOT #CIn.Straigtener.Lift_Entry.Rest;
           #Ctrl.EndOfCoil.StraightRollExit_Open := NOT #CIn.Straigtener.Lift_Exit.Rest;

           IF NOT #Ctrl.EndOfCoil.StraightRollEntry_Open
               AND
               NOT #Ctrl.EndOfCoil.StraightRollExit_Open 
           THEN
               IF #Config.MatCounter_Exist THEN
                   #Sts.EndOfCoil.Status += 1;
               ELSE
                   #Sts.EndOfCoil.Status := 10;
               END_IF;
           END_IF;

           //#######################################################################################################
           // Status = 4 - Pinch roll positioning to cut execution 
           //#######################################################################################################    
       4:



           #Ctrl.EndOfCoil.JB_Pinch_Fwd :=
           (
           NOT #Sts.EndOfCoil.Reached_TargetPosMat_TailCutExe
           AND
           NOT #Pers.Data.END_OF_COIL.Tail_ReachCutPosition
           AND
           NOT #Sts.EndOfCoil.StopPinchRoll_TargetPosMat_TailCutExe
           AND
           #Config.MatCounter_Exist
           )
           OR
           (
           NOT #Config.MatCounter_Exist
           AND
           NOT #TON_PinchrollFwd.Q
           );


           #Ctrl.EndOfCoil.Straightener_Fwd := #Ctrl.EndOfCoil.JB_Pinch_Fwd;

           IF NOT #Ctrl.EndOfCoil.JB_Pinch_Fwd THEN
               #Sts.EndOfCoil.Status += 1;
           END_IF;

           //#######################################################################################################
           // Status = 5 - Pinch roll wait standstill
           //#######################################################################################################    
       5:

           #Ctrl.EndOfCoil.JB_Pinch_Fwd := FALSE;
           #Ctrl.EndOfCoil.Straightener_Fwd := false;


           IF #CIn.JB.Pinchroll_Feed.Standstill
           THEN

               #Pers.Data.END_OF_COIL.Tail_ReachCutPosition := TRUE;
               #Sts.EndOfCoil.Status += 1;
           END_IF;


           //#######################################################################################################
           // Status = 6 - JB Cut work
           //#######################################################################################################    
       6:
           #Ctrl.EndOfCoil.JB_Pinch_Fwd := FALSE;
           #Ctrl.EndOfCoil.Straightener_Fwd := false;


           #Ctrl.EndOfCoil.JB_Cut_Work := NOT #Pers.Data.END_OF_COIL.Tail_CutDone;
           #Ctrl.EndOfCoil.JB_Cut_Rest := FALSE;

           IF #CIn.JB.CutHead.Work
           THEN
               #Pers.Data.END_OF_COIL.Tail_CutDone := TRUE;
               #Sts.EndOfCoil.Status += 1;
           END_IF;


           //#######################################################################################################
           // Status = 7 - JB Cut rest
           //#######################################################################################################    
       7:
           #Ctrl.EndOfCoil.JB_Cut_Rest := NOT #CIn.JB.CutHead.Rest;
           #Ctrl.EndOfCoil.JB_Cut_Work := FALSE;

           IF #CIn.JB.CutHead.Rest
           THEN
               #Sts.EndOfCoil.Status += 1;
           END_IF;



           //#######################################################################################################
           // Status = 8 -  Pinch roll positioning to junction position
           //#######################################################################################################    
       8:
           #Ctrl.EndOfCoil.JB_Pinch_Fwd :=
           NOT #Pers.Data.END_OF_COIL.Tail_ReachJunctionPos
           AND
           NOT #Sts.EndOfCoil.StopPinchRoll_TargetPosMat_JunctionExe
           AND
           NOT #Sts.EndOfCoil.Reached_TargetPosMat_JunctionExe
           ;


           IF NOT #Ctrl.EndOfCoil.JB_Pinch_Fwd THEN
               #Sts.EndOfCoil.Status += 1;
           END_IF;


           //#######################################################################################################
           // Status = 9 - Pinch roll wait standstill
           //#######################################################################################################    
       9:

           #Ctrl.EndOfCoil.JB_Pinch_Fwd := FALSE;

           IF #CIn.JB.Pinchroll_Feed.Standstill
           THEN
               #Pers.Data.END_OF_COIL.Tail_ReachJunctionPos := TRUE;
               #Sts.EndOfCoil.Status += 1;
           END_IF;


           //#######################################################################################################
           // Status = 10 - Decoiler 2 in position
           //#######################################################################################################
           //
       10:
           IF #CIn.DecoilersHRot.Decoiler2_InLine THEN

               #Ctrl.EndOfCoil.Decoiler_Fwd := TRUE;
               IF #DataIn.Decoiler2_PosizioneRazza THEN
                   #Ctrl.EndOfCoil.Decoiler_Fwd := FALSE;
                   #Sts.EndOfCoil.Status += 1;
               END_IF;
           ELSE
               #Ctrl.EndOfCoil.Decoiler_Fwd := FALSE;
               #Sts.EndOfCoil.Status += 1;
           END_IF;

           //#######################################################################################################
           // Status = 11 - End of sequence
           //#######################################################################################################
           //
       11:
           #Ctrl.EndOfCoil.ChangeCoilExe :=
           #Pers.Data.CoilLoadedInDecoiler1 OR
           #Pers.Data.CoilLoadedInDecoiler2;



           IF NOT #Ctrl.EndOfCoil.ChangeCoilExe
           THEN
               #Alarm.EndOfMaterial := TRUE;
               #Sts.EndOfCoil.Status += 1;
           END_IF;
           //#######################################################################################################
           // Status = 12 - End of sequence
           //#######################################################################################################
           //
       12:
           ;
           //#######################################################################################################
           // Status = 99 - Abort
           //#######################################################################################################       
       99:

           IF NOT #Alarm.S_MatPresence_StraightExit_NotOFF
           THEN
               #Sts.EndOfCoil.Status := 0;
           END_IF;


   END_CASE;
END_REGION

REGION Network 54 (SCL): End of coil - Sequence 2 Cut Tail



   CASE #Sts.EndOfCoil.Status OF

           //#######################################################################################################
           // Status = 20 - Fwd Pinchroll + Straightener 
           //#######################################################################################################    

       20:

           #Ctrl.EndOfCoil.JB_Pinch_Fwd := #Pers.Data.MaterialPresence_StraightenerExit;
           #Ctrl.EndOfCoil.Straightener_Fwd := #Ctrl.EndOfCoil.JB_Pinch_Fwd;

           IF #TON_StraightnerFwd.Q OR
               NOT #Pers.Data.MaterialPresence_StraightenerEntry
           THEN
               #Ctrl.EndOfCoil.Straightener_Fwd := FALSE;
               #Ctrl.EndOfCoil.JB_Pinch_Fwd := FALSE;
               #Sts.EndOfCoil.Status += 1;
           END_IF;

           //#######################################################################################################
           // Status = 21 - Wait standstill
           //#######################################################################################################    

       21:

           #Ctrl.EndOfCoil.JB_Pinch_Fwd := FALSE;
           #Ctrl.EndOfCoil.Straightener_Fwd := FALSE;

           IF #CIn.JB.Pinchroll_Feed.Standstill AND
               #CIn.Straigtener.Feed.Standstill
           THEN
               #Sts.EndOfCoil.Status += 1;
           END_IF;


           //#######################################################################################################
           // Status = 22 - JB Cut work
           //#######################################################################################################    
       22:
           #Ctrl.EndOfCoil.JB_Pinch_Fwd := FALSE;
           #Ctrl.EndOfCoil.Straightener_Fwd := FALSE;


           #Ctrl.EndOfCoil.JB_Cut_Work := NOT #Pers.Data.END_OF_COIL.Tail_CutDone;
           #Ctrl.EndOfCoil.JB_Cut_Rest := FALSE;

           IF #CIn.JB.CutHead.Work
           THEN
               #Pers.Data.END_OF_COIL.SaveEncPosMat_CutDone := #CIn.MaterialCounter.Data.CounterValue;
               #Pers.Data.END_OF_COIL.Tail_CutDone := TRUE;
               #Sts.EndOfCoil.Status += 1;
           END_IF;

           //#######################################################################################################
           // Status = 23 - JB Cut rest
           //#######################################################################################################    
       23:
           #Ctrl.EndOfCoil.JB_Cut_Rest := NOT #CIn.JB.CutHead.Rest;
           #Ctrl.EndOfCoil.JB_Cut_Work := FALSE;

           IF #CIn.JB.CutHead.Rest
           THEN
               #Sts.EndOfCoil.Status += 1;
           END_IF;


           //#######################################################################################################
           // Status = 24 - Straightner Bwd
           //#######################################################################################################    

       24:

           #Ctrl.EndOfCoil.Straightener_Bwd := TRUE;

           IF #TON_StraightnerBwd.Q THEN
               #Ctrl.EndOfCoil.Straightener_Bwd := FALSE;
               #Sts.EndOfCoil.Status += 1;
           END_IF;


           //#######################################################################################################
           // Status = 25 - Open rolls of straightener
           //#######################################################################################################    
       25:

           #Ctrl.EndOfCoil.StraightRollEntry_Open := NOT #CIn.Straigtener.Lift_Entry.Rest;
           #Ctrl.EndOfCoil.StraightRollExit_Open := NOT #CIn.Straigtener.Lift_Exit.Rest;

           IF NOT #Ctrl.EndOfCoil.StraightRollEntry_Open
               AND
               NOT #Ctrl.EndOfCoil.StraightRollExit_Open
           THEN
               IF #Config.MatCounter_Exist THEN
                   #Sts.EndOfCoil.Status := 8;
               ELSE
                   #Sts.EndOfCoil.Status := 10;
               END_IF;
           END_IF;



   END_CASE;
END_REGION

REGION Network 55: <<+>>
END_REGION

REGION Network 56: <<+>>
END_REGION

REGION Network 57 (SCL): Thickness control function - Coordination in
   //
   #ThicknessCheck.CIn.Rst := #AreaInterface.RstAlarms;
   //
   #ThicknessCheck.CIn.Init :=
   NOT (
   #Pers.Data.MaterialPresence_StraightenerEntry
   AND
   #Pers.Data.MaterialPresence_StraightenerExit
   AND
   #Pers.Data.MaterialPresence_JBPinchExit
   AND
   NOT #Pers.Data.MATERIAL_SEPARATION.Mem
   AND
   NOT
   #Pers.Data.END_OF_COIL.Mem
   );

   //
   #ThicknessCheck.CIn.Enable := 
   NOT #ThicknessCheck.CIn.Init
   AND
   #CIn.MaterialCounter.Data.CounterValid
   AND
   "PPrf_MAIN".ON_WORK.GeneralData.Material_Thickness > 0.0;
   //
   #ThicknessCheck.CIn.MaterialCounter := #CIn.MaterialCounter.Data.CounterValue;
   //
   #ThicknessCheck.CIn.Setpoint := "PPrf_MAIN".ON_WORK.GeneralData.Material_Thickness;


   #ThicknessCheck.CIn.Init := #HMI.ThicknessControl.Button_Init;
END_REGION

REGION Network 58: Thickness control function
   RUNG wire#powerrail
      #ThicknessCheck("HW_ID_DL-PN" := #"ThicknessCheck_HW_ID_DL-PN", HW_ID_IL1000 := #ThicknessCheck_HW_ID_IL1000, HW_ID_IL1050 := #ThicknessCheck_HW_ID_IL1050, CIn :=, HMI := #HMI.ThicknessControl, Par := #Pers.Par.Thickness, Pers_Data := #Pers.Data.Thickness, Alarm := #Alarm.TichnessCheck, Warning := #Warning.ThicnessCheck, Cout =>)
   END_RUNG
   // the same network as SCL:
   #ThicknessCheck("HW_ID_DL-PN" := #"ThicknessCheck_HW_ID_DL-PN",   // "ThicknessCheck_FB"
                   HW_ID_IL1000 := #ThicknessCheck_HW_ID_IL1000,
                   HW_ID_IL1050 := #ThicknessCheck_HW_ID_IL1050,
                   HMI := #HMI.ThicknessControl,
                   Par := #Pers.Par.Thickness,
                   Pers_Data := #Pers.Data.Thickness,
                   Alarm := #Alarm.TichnessCheck,
                   Warning := #Warning.ThicnessCheck);
END_REGION

REGION Network 59: <<+>>
END_REGION

REGION Network 60: <<+>>
END_REGION

REGION Network 61: MES
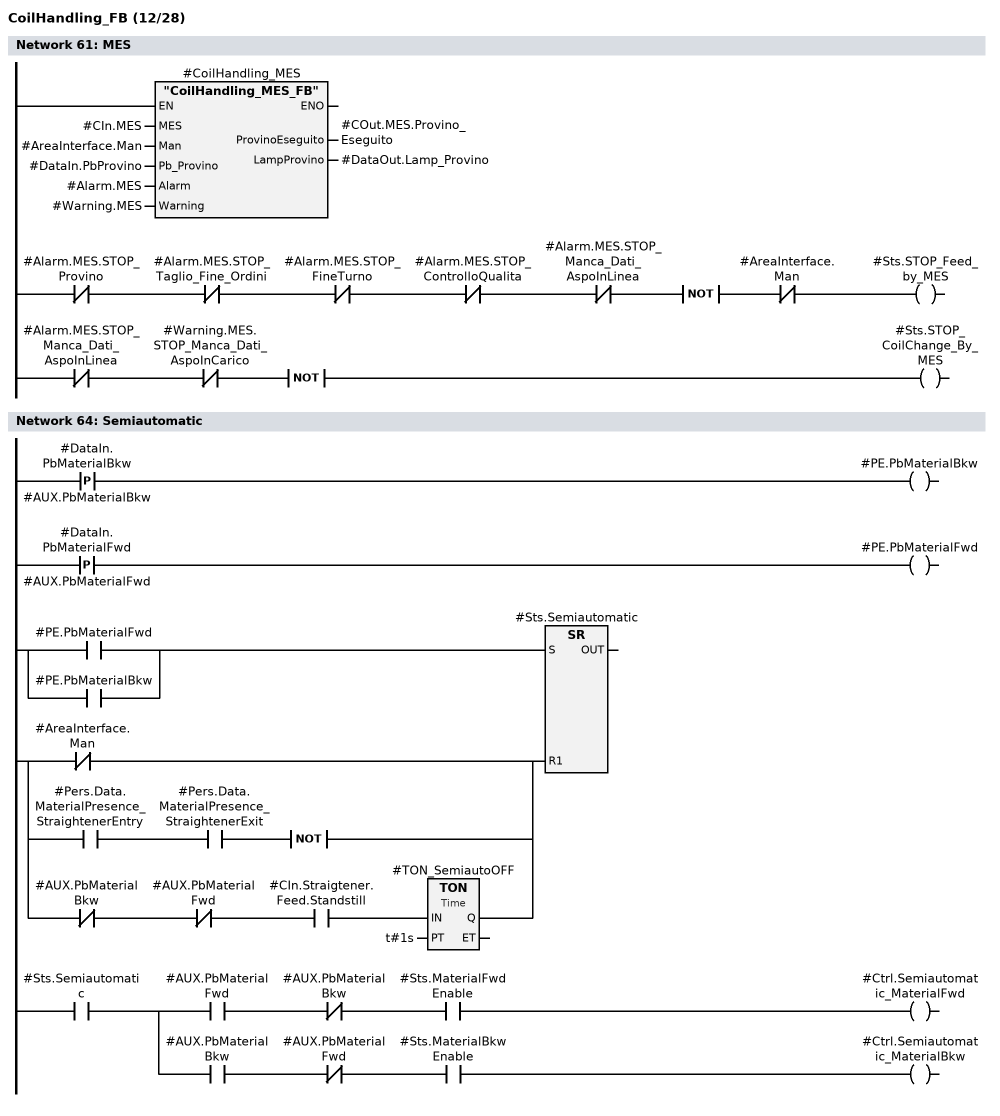
   RUNG wire#powerrail
      #CoilHandling_MES(MES := #CIn.MES, Man := #AreaInterface.Man, Pb_Provino := #DataIn.PbProvino, Alarm := #Alarm.MES, Warning := #Warning.MES, ProvinoEseguito => #COut.MES.Provino_Eseguito, LampProvino => #DataOut.Lamp_Provino)
   END_RUNG
   RUNG wire#powerrail
      I_Contact( #Alarm.MES.STOP_Provino )
      I_Contact( #Alarm.MES.STOP_Taglio_Fine_Ordini )
      I_Contact( #Alarm.MES.STOP_FineTurno )
      I_Contact( #Alarm.MES.STOP_ControlloQualita )
      I_Contact( #Alarm.MES.STOP_Manca_Dati_AspoInLinea )
      Not()
      I_Contact( #AreaInterface.Man )
      Coil( #Sts.STOP_Feed_by_MES )
   END_RUNG
   RUNG wire#powerrail
      I_Contact( #Alarm.MES.STOP_Manca_Dati_AspoInLinea )
      I_Contact( #Warning.MES.STOP_Manca_Dati_AspoInCarico )
      Not()
      Coil( #Sts.STOP_CoilChange_By_MES )
   END_RUNG
   // the same network as SCL:
   #CoilHandling_MES(MES := #CIn.MES,   // "CoilHandling_MES_FB"
                     Man := #AreaInterface.Man,
                     Pb_Provino := #DataIn.PbProvino,
                     Alarm := #Alarm.MES,
                     Warning := #Warning.MES,
                     ProvinoEseguito => #COut.MES.Provino_Eseguito,
                     LampProvino => #DataOut.Lamp_Provino);
   #Sts.STOP_Feed_by_MES := NOT (NOT #Alarm.MES.STOP_Provino AND NOT #Alarm.MES.STOP_Taglio_Fine_Ordini AND NOT #Alarm.MES.STOP_FineTurno AND NOT #Alarm.MES.STOP_ControlloQualita AND NOT #Alarm.MES.STOP_Manca_Dati_AspoInLinea) AND NOT #AreaInterface.Man;
   #Sts.STOP_CoilChange_By_MES := NOT (NOT #Alarm.MES.STOP_Manca_Dati_AspoInLinea AND NOT #Warning.MES.STOP_Manca_Dati_AspoInCarico);
END_REGION

REGION Network 62: <<+>>
END_REGION

REGION Network 63: <<+>>
END_REGION

REGION Network 64: Semiautomatic
   RUNG wire#powerrail
      P_Contact(operand := #DataIn.PbMaterialBkw, bit := #AUX.PbMaterialBkw)
      Coil( #PE.PbMaterialBkw )
   END_RUNG
   RUNG wire#powerrail
      P_Contact(operand := #DataIn.PbMaterialFwd, bit := #AUX.PbMaterialFwd)
      Coil( #PE.PbMaterialFwd )
   END_RUNG
   RUNG wire#powerrail
      Contact( #PE.PbMaterialFwd )
      wire#w1
      S_SR(operand := #Sts.Semiautomatic, r1 := wire#w2)
   END_RUNG
   RUNG wire#powerrail
      Contact( #PE.PbMaterialBkw )
   END_RUNG wire#w1
   RUNG wire#powerrail
      I_Contact( #AreaInterface.Man )
   END_RUNG wire#w2
   RUNG wire#powerrail
      Contact( #Pers.Data.MaterialPresence_StraightenerEntry )
      Contact( #Pers.Data.MaterialPresence_StraightenerExit )
      Not()
   END_RUNG wire#w2
   RUNG wire#powerrail
      I_Contact( #AUX.PbMaterialBkw )
      I_Contact( #AUX.PbMaterialFwd )
      Contact( #CIn.Straigtener.Feed.Standstill )
      { S7_Templates := "time_type := Time" } #TON_SemiautoOFF.TON(pt := t#1s, et =>)
   END_RUNG wire#w2
   RUNG wire#powerrail
      Contact( #Sts.Semiautomatic )
      wire#w3
      Contact( #AUX.PbMaterialFwd )
      I_Contact( #AUX.PbMaterialBkw )
      Contact( #Sts.MaterialFwdEnable )
      Coil( #Ctrl.Semiautomatic_MaterialFwd )
   END_RUNG
   RUNG wire#w3
      Contact( #AUX.PbMaterialBkw )
      I_Contact( #AUX.PbMaterialFwd )
      Contact( #Sts.MaterialBkwEnable )
      Coil( #Ctrl.Semiautomatic_MaterialBkw )
   END_RUNG
   // the same network as SCL:
   #_w1 := #DataIn.PbMaterialBkw AND NOT #AUX.PbMaterialBkw;   // rising edge of #DataIn.PbMaterialBkw
   #AUX.PbMaterialBkw := #DataIn.PbMaterialBkw;
   #PE.PbMaterialBkw := #_w1;
   #_w2 := #DataIn.PbMaterialFwd AND NOT #AUX.PbMaterialFwd;   // rising edge of #DataIn.PbMaterialFwd
   #AUX.PbMaterialFwd := #DataIn.PbMaterialFwd;
   #PE.PbMaterialFwd := #_w2;
   #TON_SemiautoOFF(IN := NOT #AUX.PbMaterialBkw AND NOT #AUX.PbMaterialFwd AND #CIn.Straigtener.Feed.Standstill,   // TON
                    PT := t#1s);
   IF #PE.PbMaterialFwd OR #PE.PbMaterialBkw THEN
       #Sts.Semiautomatic := TRUE;   // SR flip-flop
   END_IF;
   IF NOT #AreaInterface.Man OR NOT (#Pers.Data.MaterialPresence_StraightenerEntry AND #Pers.Data.MaterialPresence_StraightenerExit) OR #TON_SemiautoOFF.Q THEN
       #Sts.Semiautomatic := FALSE;
   END_IF;
   #Ctrl.Semiautomatic_MaterialFwd := #Sts.Semiautomatic AND #AUX.PbMaterialFwd AND NOT #AUX.PbMaterialBkw AND #Sts.MaterialFwdEnable;
   #Ctrl.Semiautomatic_MaterialBkw := #Sts.Semiautomatic AND #AUX.PbMaterialBkw AND NOT #AUX.PbMaterialFwd AND #Sts.MaterialBkwEnable;
END_REGION

REGION Network 65: Semiautomatic material BWD
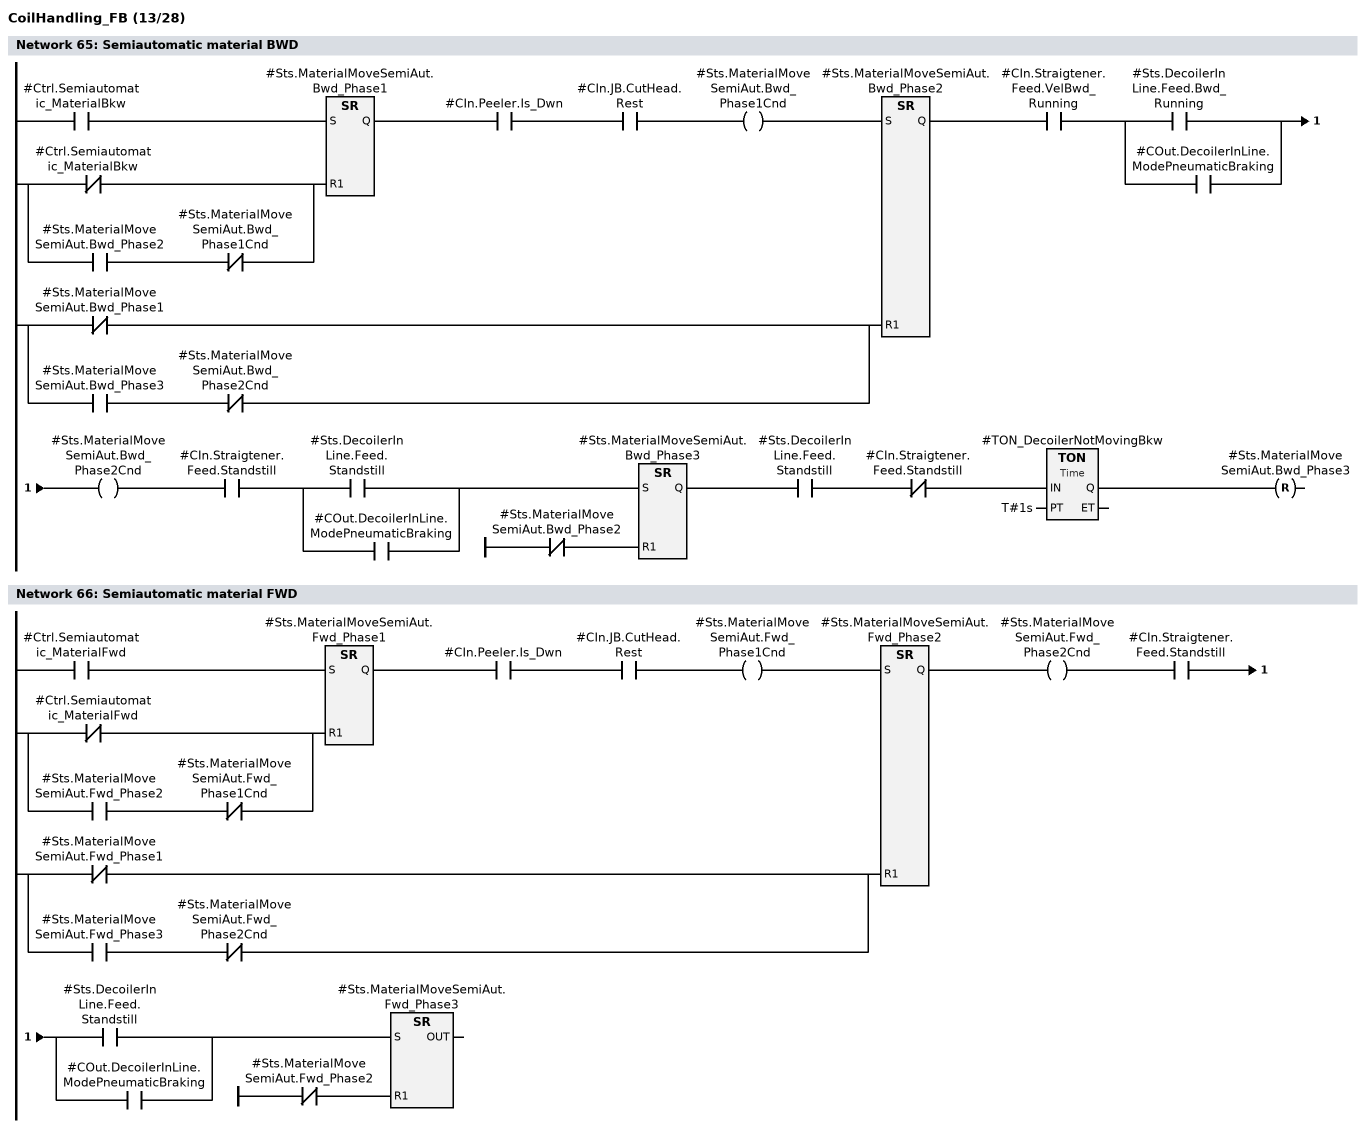
   RUNG wire#powerrail
      Contact( #Ctrl.Semiautomatic_MaterialBkw )
      S_SR(operand := #Sts.MaterialMoveSemiAut.Bwd_Phase1, r1 := wire#w1)
      Contact( #CIn.Peeler.Is_Dwn )
      Contact( #CIn.JB.CutHead.Rest )
      Coil( #Sts.MaterialMoveSemiAut.Bwd_Phase1Cnd )
      S_SR(operand := #Sts.MaterialMoveSemiAut.Bwd_Phase2, r1 := wire#w2)
      Contact( #CIn.Straigtener.Feed.VelBwd_Running )
      wire#w3
      Contact( #Sts.DecoilerInLine.Feed.Bwd_Running )
      wire#w4
      Coil( #Sts.MaterialMoveSemiAut.Bwd_Phase2Cnd )
      Contact( #CIn.Straigtener.Feed.Standstill )
      wire#w5
      Contact( #Sts.DecoilerInLine.Feed.Standstill )
      wire#w6
      S_SR(operand := #Sts.MaterialMoveSemiAut.Bwd_Phase3, r1 := wire#w7)
      Contact( #Sts.DecoilerInLine.Feed.Standstill )
      I_Contact( #CIn.Straigtener.Feed.Standstill )
      { S7_Templates := "time_type := Time" } #TON_DecoilerNotMovingBkw.TON(pt := T#1s, et =>)
      R_Coil( #Sts.MaterialMoveSemiAut.Bwd_Phase3 )
   END_RUNG
   RUNG wire#powerrail
      I_Contact( #Ctrl.Semiautomatic_MaterialBkw )
   END_RUNG wire#w1
   RUNG wire#powerrail
      Contact( #Sts.MaterialMoveSemiAut.Bwd_Phase2 )
      I_Contact( #Sts.MaterialMoveSemiAut.Bwd_Phase1Cnd )
   END_RUNG wire#w1
   RUNG wire#powerrail
      I_Contact( #Sts.MaterialMoveSemiAut.Bwd_Phase1 )
   END_RUNG wire#w2
   RUNG wire#powerrail
      Contact( #Sts.MaterialMoveSemiAut.Bwd_Phase3 )
      I_Contact( #Sts.MaterialMoveSemiAut.Bwd_Phase2Cnd )
   END_RUNG wire#w2
   RUNG wire#w3
      Contact( #COut.DecoilerInLine.ModePneumaticBraking )
   END_RUNG wire#w4
   RUNG wire#w5
      Contact( #COut.DecoilerInLine.ModePneumaticBraking )
   END_RUNG wire#w6
   RUNG wire#powerrail
      I_Contact( #Sts.MaterialMoveSemiAut.Bwd_Phase2 )
   END_RUNG wire#w7
   // the same network as SCL:
   IF #Ctrl.Semiautomatic_MaterialBkw THEN
       #Sts.MaterialMoveSemiAut.Bwd_Phase1 := TRUE;   // SR flip-flop
   END_IF;
   IF NOT #Ctrl.Semiautomatic_MaterialBkw OR (#Sts.MaterialMoveSemiAut.Bwd_Phase2 AND NOT #Sts.MaterialMoveSemiAut.Bwd_Phase1Cnd) THEN
       #Sts.MaterialMoveSemiAut.Bwd_Phase1 := FALSE;
   END_IF;
   #Sts.MaterialMoveSemiAut.Bwd_Phase1Cnd := #Sts.MaterialMoveSemiAut.Bwd_Phase1 AND #CIn.Peeler.Is_Dwn AND #CIn.JB.CutHead.Rest;
   IF #Sts.MaterialMoveSemiAut.Bwd_Phase1Cnd THEN
       #Sts.MaterialMoveSemiAut.Bwd_Phase2 := TRUE;   // SR flip-flop
   END_IF;
   IF NOT #Sts.MaterialMoveSemiAut.Bwd_Phase1 OR (#Sts.MaterialMoveSemiAut.Bwd_Phase3 AND NOT #Sts.MaterialMoveSemiAut.Bwd_Phase2Cnd) THEN
       #Sts.MaterialMoveSemiAut.Bwd_Phase2 := FALSE;
   END_IF;
   #Sts.MaterialMoveSemiAut.Bwd_Phase2Cnd := #Sts.MaterialMoveSemiAut.Bwd_Phase2 AND #CIn.Straigtener.Feed.VelBwd_Running AND (#Sts.DecoilerInLine.Feed.Bwd_Running OR #COut.DecoilerInLine.ModePneumaticBraking);
   IF #Sts.MaterialMoveSemiAut.Bwd_Phase2Cnd AND #CIn.Straigtener.Feed.Standstill AND (#Sts.DecoilerInLine.Feed.Standstill OR #COut.DecoilerInLine.ModePneumaticBraking) THEN
       #Sts.MaterialMoveSemiAut.Bwd_Phase3 := TRUE;   // SR flip-flop
   END_IF;
   IF NOT #Sts.MaterialMoveSemiAut.Bwd_Phase2 THEN #Sts.MaterialMoveSemiAut.Bwd_Phase3 := FALSE; END_IF;
   #TON_DecoilerNotMovingBkw(IN := #Sts.MaterialMoveSemiAut.Bwd_Phase3 AND #Sts.DecoilerInLine.Feed.Standstill AND NOT #CIn.Straigtener.Feed.Standstill,   // TON
                           PT := T#1s);
   IF #TON_DecoilerNotMovingBkw.Q THEN #Sts.MaterialMoveSemiAut.Bwd_Phase3 := FALSE; END_IF;
END_REGION

REGION Network 66: Semiautomatic material FWD
   RUNG wire#powerrail
      Contact( #Ctrl.Semiautomatic_MaterialFwd )
      S_SR(operand := #Sts.MaterialMoveSemiAut.Fwd_Phase1, r1 := wire#w1)
      Contact( #CIn.Peeler.Is_Dwn )
      Contact( #CIn.JB.CutHead.Rest )
      Coil( #Sts.MaterialMoveSemiAut.Fwd_Phase1Cnd )
      S_SR(operand := #Sts.MaterialMoveSemiAut.Fwd_Phase2, r1 := wire#w2)
      Coil( #Sts.MaterialMoveSemiAut.Fwd_Phase2Cnd )
      Contact( #CIn.Straigtener.Feed.Standstill )
      wire#w3
      Contact( #Sts.DecoilerInLine.Feed.Standstill )
      wire#w4
      S_SR(operand := #Sts.MaterialMoveSemiAut.Fwd_Phase3, r1 := wire#w5)
   END_RUNG
   RUNG wire#powerrail
      I_Contact( #Ctrl.Semiautomatic_MaterialFwd )
   END_RUNG wire#w1
   RUNG wire#powerrail
      Contact( #Sts.MaterialMoveSemiAut.Fwd_Phase2 )
      I_Contact( #Sts.MaterialMoveSemiAut.Fwd_Phase1Cnd )
   END_RUNG wire#w1
   RUNG wire#powerrail
      I_Contact( #Sts.MaterialMoveSemiAut.Fwd_Phase1 )
   END_RUNG wire#w2
   RUNG wire#powerrail
      Contact( #Sts.MaterialMoveSemiAut.Fwd_Phase3 )
      I_Contact( #Sts.MaterialMoveSemiAut.Fwd_Phase2Cnd )
   END_RUNG wire#w2
   RUNG wire#w3
      Contact( #COut.DecoilerInLine.ModePneumaticBraking )
   END_RUNG wire#w4
   RUNG wire#powerrail
      I_Contact( #Sts.MaterialMoveSemiAut.Fwd_Phase2 )
   END_RUNG wire#w5
   // the same network as SCL:
   IF #Ctrl.Semiautomatic_MaterialFwd THEN
       #Sts.MaterialMoveSemiAut.Fwd_Phase1 := TRUE;   // SR flip-flop
   END_IF;
   IF NOT #Ctrl.Semiautomatic_MaterialFwd OR (#Sts.MaterialMoveSemiAut.Fwd_Phase2 AND NOT #Sts.MaterialMoveSemiAut.Fwd_Phase1Cnd) THEN
       #Sts.MaterialMoveSemiAut.Fwd_Phase1 := FALSE;
   END_IF;
   #Sts.MaterialMoveSemiAut.Fwd_Phase1Cnd := #Sts.MaterialMoveSemiAut.Fwd_Phase1 AND #CIn.Peeler.Is_Dwn AND #CIn.JB.CutHead.Rest;
   IF #Sts.MaterialMoveSemiAut.Fwd_Phase1Cnd THEN
       #Sts.MaterialMoveSemiAut.Fwd_Phase2 := TRUE;   // SR flip-flop
   END_IF;
   IF NOT #Sts.MaterialMoveSemiAut.Fwd_Phase1 OR (#Sts.MaterialMoveSemiAut.Fwd_Phase3 AND NOT #Sts.MaterialMoveSemiAut.Fwd_Phase2Cnd) THEN
       #Sts.MaterialMoveSemiAut.Fwd_Phase2 := FALSE;
   END_IF;
   #Sts.MaterialMoveSemiAut.Fwd_Phase2Cnd := #Sts.MaterialMoveSemiAut.Fwd_Phase2;
   IF #Sts.MaterialMoveSemiAut.Fwd_Phase2 AND #CIn.Straigtener.Feed.Standstill AND (#Sts.DecoilerInLine.Feed.Standstill OR #COut.DecoilerInLine.ModePneumaticBraking) THEN
       #Sts.MaterialMoveSemiAut.Fwd_Phase3 := TRUE;   // SR flip-flop
   END_IF;
   IF NOT #Sts.MaterialMoveSemiAut.Fwd_Phase2 THEN #Sts.MaterialMoveSemiAut.Fwd_Phase3 := FALSE; END_IF;
END_REGION

REGION Network 67: <<+>>
END_REGION

REGION Network 68: Automatic material FWD
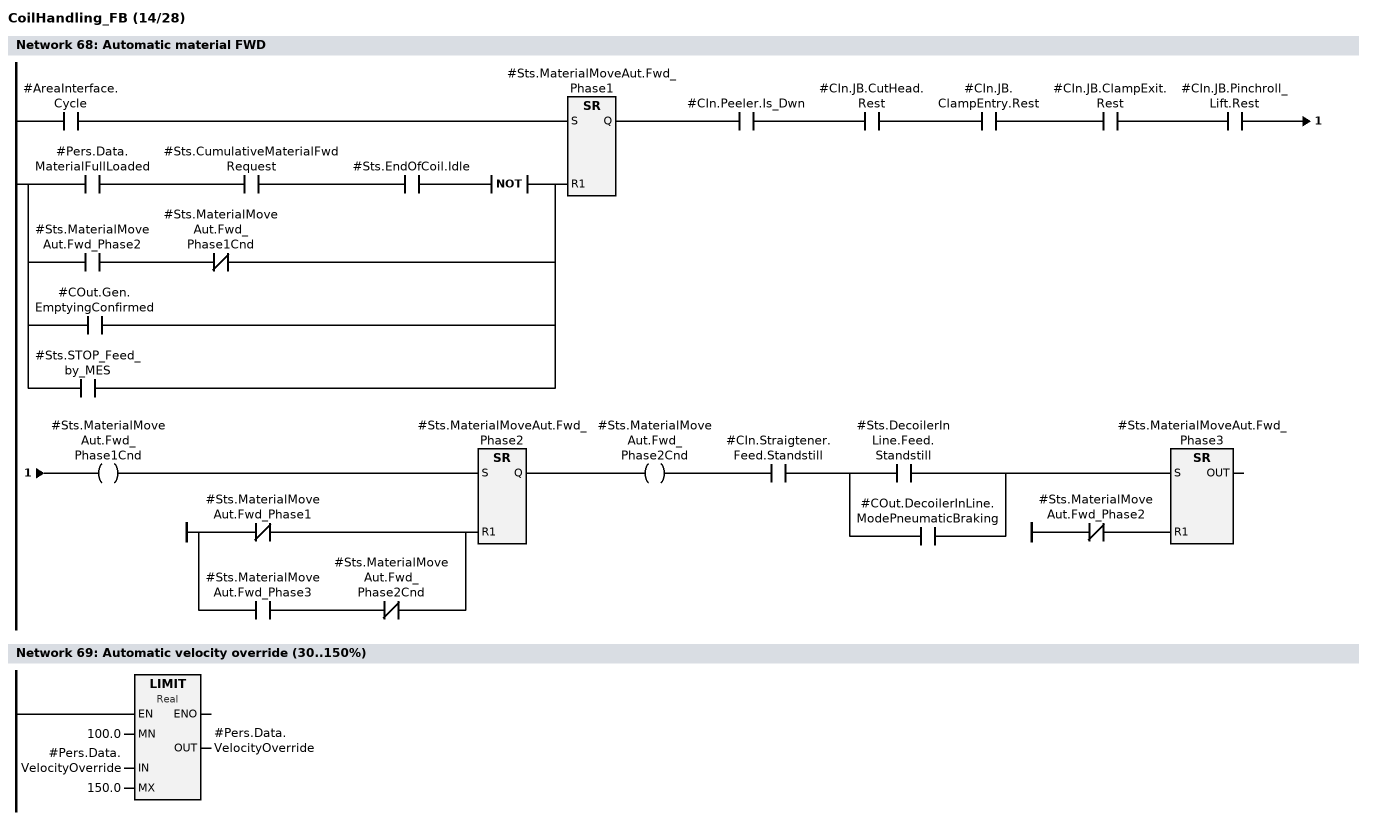
   RUNG wire#powerrail
      Contact( #AreaInterface.Cycle )
      S_SR(operand := #Sts.MaterialMoveAut.Fwd_Phase1, r1 := wire#w1)
      Contact( #CIn.Peeler.Is_Dwn )
      Contact( #CIn.JB.CutHead.Rest )
      Contact( #CIn.JB.ClampEntry.Rest )
      Contact( #CIn.JB.ClampExit.Rest )
      Contact( #CIn.JB.Pinchroll_Lift.Rest )
      Coil( #Sts.MaterialMoveAut.Fwd_Phase1Cnd )
      S_SR(operand := #Sts.MaterialMoveAut.Fwd_Phase2, r1 := wire#w2)
      Coil( #Sts.MaterialMoveAut.Fwd_Phase2Cnd )
      Contact( #CIn.Straigtener.Feed.Standstill )
      wire#w3
      Contact( #Sts.DecoilerInLine.Feed.Standstill )
      wire#w4
      S_SR(operand := #Sts.MaterialMoveAut.Fwd_Phase3, r1 := wire#w5)
   END_RUNG
   RUNG wire#powerrail
      Contact( #Pers.Data.MaterialFullLoaded )
      Contact( #Sts.CumulativeMaterialFwdRequest )
      Contact( #Sts.EndOfCoil.Idle )
      Not()
   END_RUNG wire#w1
   RUNG wire#powerrail
      Contact( #Sts.MaterialMoveAut.Fwd_Phase2 )
      I_Contact( #Sts.MaterialMoveAut.Fwd_Phase1Cnd )
   END_RUNG wire#w1
   RUNG wire#powerrail
      Contact( #COut.Gen.EmptyingConfirmed )
   END_RUNG wire#w1
   RUNG wire#powerrail
      Contact( #Sts.STOP_Feed_by_MES )
   END_RUNG wire#w1
   RUNG wire#powerrail
      I_Contact( #Sts.MaterialMoveAut.Fwd_Phase1 )
   END_RUNG wire#w2
   RUNG wire#powerrail
      Contact( #Sts.MaterialMoveAut.Fwd_Phase3 )
      I_Contact( #Sts.MaterialMoveAut.Fwd_Phase2Cnd )
   END_RUNG wire#w2
   RUNG wire#w3
      Contact( #COut.DecoilerInLine.ModePneumaticBraking )
   END_RUNG wire#w4
   RUNG wire#powerrail
      I_Contact( #Sts.MaterialMoveAut.Fwd_Phase2 )
   END_RUNG wire#w5
   // the same network as SCL:
   IF #AreaInterface.Cycle THEN
       #Sts.MaterialMoveAut.Fwd_Phase1 := TRUE;   // SR flip-flop
   END_IF;
   IF NOT (#Pers.Data.MaterialFullLoaded AND #Sts.CumulativeMaterialFwdRequest AND #Sts.EndOfCoil.Idle) OR (#Sts.MaterialMoveAut.Fwd_Phase2 AND NOT #Sts.MaterialMoveAut.Fwd_Phase1Cnd) OR #COut.Gen.EmptyingConfirmed OR #Sts.STOP_Feed_by_MES THEN
       #Sts.MaterialMoveAut.Fwd_Phase1 := FALSE;
   END_IF;
   #Sts.MaterialMoveAut.Fwd_Phase1Cnd := #Sts.MaterialMoveAut.Fwd_Phase1 AND #CIn.Peeler.Is_Dwn AND #CIn.JB.CutHead.Rest AND #CIn.JB.ClampEntry.Rest AND #CIn.JB.ClampExit.Rest AND #CIn.JB.Pinchroll_Lift.Rest;
   IF #Sts.MaterialMoveAut.Fwd_Phase1Cnd THEN
       #Sts.MaterialMoveAut.Fwd_Phase2 := TRUE;   // SR flip-flop
   END_IF;
   IF NOT #Sts.MaterialMoveAut.Fwd_Phase1 OR (#Sts.MaterialMoveAut.Fwd_Phase3 AND NOT #Sts.MaterialMoveAut.Fwd_Phase2Cnd) THEN
       #Sts.MaterialMoveAut.Fwd_Phase2 := FALSE;
   END_IF;
   #Sts.MaterialMoveAut.Fwd_Phase2Cnd := #Sts.MaterialMoveAut.Fwd_Phase2;
   IF #Sts.MaterialMoveAut.Fwd_Phase2 AND #CIn.Straigtener.Feed.Standstill AND (#Sts.DecoilerInLine.Feed.Standstill OR #COut.DecoilerInLine.ModePneumaticBraking) THEN
       #Sts.MaterialMoveAut.Fwd_Phase3 := TRUE;   // SR flip-flop
   END_IF;
   IF NOT #Sts.MaterialMoveAut.Fwd_Phase2 THEN #Sts.MaterialMoveAut.Fwd_Phase3 := FALSE; END_IF;
END_REGION

REGION Network 69: Automatic velocity override (30..150%)
   RUNG wire#powerrail
      { S7_Templates := "value_type := Real" } Limit(mn := 100.0, in := #Pers.Data.VelocityOverride, mx := 150.0, out => #Pers.Data.VelocityOverride)
   END_RUNG
   // the same network as SCL:
   #Pers.Data.VelocityOverride := LIMIT(MN := 100.0, IN := #Pers.Data.VelocityOverride, MX := 150.0);
END_REGION

REGION Network 70: <<+>>
END_REGION

REGION Network 71: Stop Inactivity
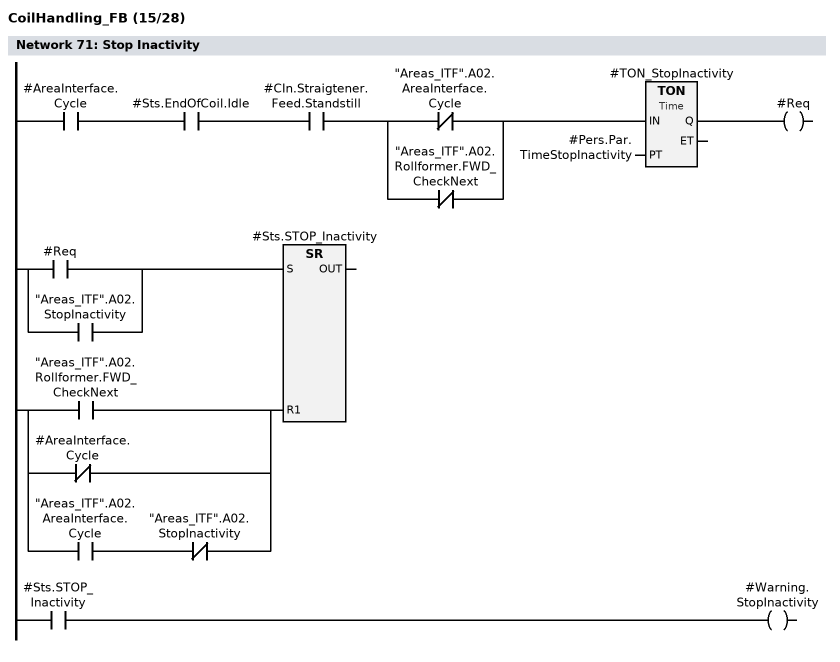
   RUNG wire#powerrail
      Contact( #AreaInterface.Cycle )
      Contact( #Sts.EndOfCoil.Idle )
      Contact( #CIn.Straigtener.Feed.Standstill )
      wire#w1
      I_Contact( "Areas_ITF".A02.AreaInterface.Cycle )
      wire#w2
      { S7_Templates := "time_type := Time" } #TON_StopInactivity.TON(pt := #Pers.Par.TimeStopInactivity, et =>)
      Coil( #Req )
   END_RUNG
   RUNG wire#w1
      I_Contact( "Areas_ITF".A02.Rollformer.FWD_CheckNext )
   END_RUNG wire#w2
   RUNG wire#powerrail
      Contact( #Req )
      wire#w3
      S_SR(operand := #Sts.STOP_Inactivity, r1 := wire#w4)
   END_RUNG
   RUNG wire#powerrail
      Contact( "Areas_ITF".A02.StopInactivity )
   END_RUNG wire#w3
   RUNG wire#powerrail
      Contact( "Areas_ITF".A02.Rollformer.FWD_CheckNext )
   END_RUNG wire#w4
   RUNG wire#powerrail
      I_Contact( #AreaInterface.Cycle )
   END_RUNG wire#w4
   RUNG wire#powerrail
      Contact( "Areas_ITF".A02.AreaInterface.Cycle )
      I_Contact( "Areas_ITF".A02.StopInactivity )
   END_RUNG wire#w4
   RUNG wire#powerrail
      Contact( #Sts.STOP_Inactivity )
      Coil( #Warning.StopInactivity )
   END_RUNG
   // the same network as SCL:
   #TON_StopInactivity(IN := #AreaInterface.Cycle AND #Sts.EndOfCoil.Idle AND #CIn.Straigtener.Feed.Standstill AND (NOT "Areas_ITF".A02.AreaInterface.Cycle OR NOT "Areas_ITF".A02.Rollformer.FWD_CheckNext),   // TON
                       PT := #Pers.Par.TimeStopInactivity);
   #Req := #TON_StopInactivity.Q;
   IF #Req OR "Areas_ITF".A02.StopInactivity THEN
       #Sts.STOP_Inactivity := TRUE;   // SR flip-flop
   END_IF;
   IF "Areas_ITF".A02.Rollformer.FWD_CheckNext OR NOT #AreaInterface.Cycle OR ("Areas_ITF".A02.AreaInterface.Cycle AND NOT "Areas_ITF".A02.StopInactivity) THEN
       #Sts.STOP_Inactivity := FALSE;
   END_IF;
   #Warning.StopInactivity := #Sts.STOP_Inactivity;
END_REGION

REGION Network 72: <<+>>
END_REGION

REGION Network 73: <<+>>
END_REGION

REGION Network 74: Coordination Out - Gen
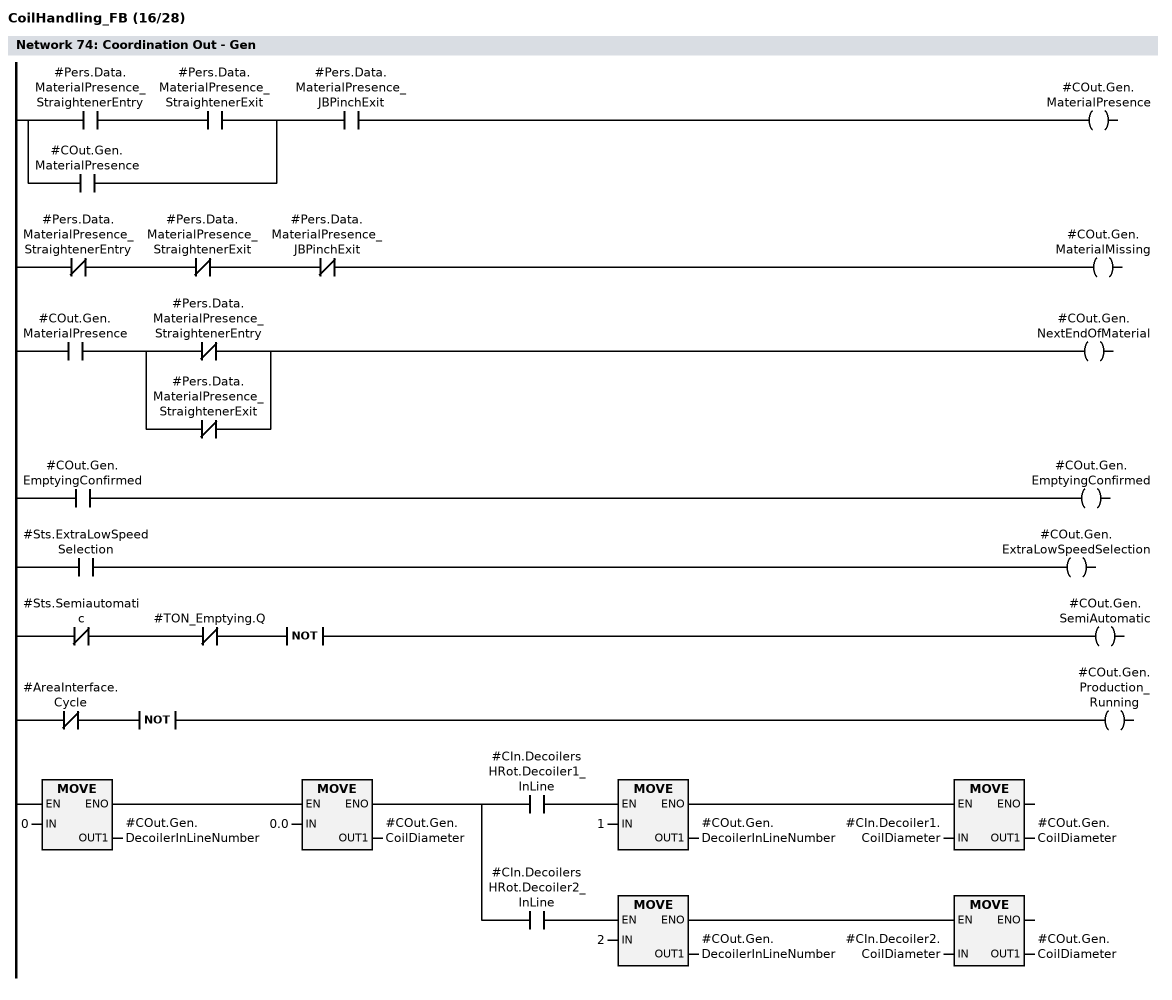
   RUNG wire#powerrail
      Contact( #Pers.Data.MaterialPresence_StraightenerEntry )
      Contact( #Pers.Data.MaterialPresence_StraightenerExit )
      wire#w1
      Contact( #Pers.Data.MaterialPresence_JBPinchExit )
      Coil( #COut.Gen.MaterialPresence )
   END_RUNG
   RUNG wire#powerrail
      Contact( #COut.Gen.MaterialPresence )
   END_RUNG wire#w1
   RUNG wire#powerrail
      I_Contact( #Pers.Data.MaterialPresence_StraightenerEntry )
      I_Contact( #Pers.Data.MaterialPresence_StraightenerExit )
      I_Contact( #Pers.Data.MaterialPresence_JBPinchExit )
      Coil( #COut.Gen.MaterialMissing )
   END_RUNG
   RUNG wire#powerrail
      Contact( #COut.Gen.MaterialPresence )
      wire#w2
      I_Contact( #Pers.Data.MaterialPresence_StraightenerEntry )
      wire#w3
      Coil( #COut.Gen.NextEndOfMaterial )
   END_RUNG
   RUNG wire#w2
      I_Contact( #Pers.Data.MaterialPresence_StraightenerExit )
   END_RUNG wire#w3
   RUNG wire#powerrail
      Contact( #COut.Gen.EmptyingConfirmed )
      Coil( #COut.Gen.EmptyingConfirmed )
   END_RUNG
   RUNG wire#powerrail
      Contact( #Sts.ExtraLowSpeedSelection )
      Coil( #COut.Gen.ExtraLowSpeedSelection )
   END_RUNG
   RUNG wire#powerrail
      I_Contact( #Sts.Semiautomatic )
      I_Contact( #TON_Emptying.Q )
      Not()
      Coil( #COut.Gen.SemiAutomatic )
   END_RUNG
   RUNG wire#powerrail
      I_Contact( #AreaInterface.Cycle )
      Not()
      Coil( #COut.Gen.Production_Running )
   END_RUNG
   RUNG wire#powerrail
      Move(in := 0, out1 => #COut.Gen.DecoilerInLineNumber)
      Move(in := 0.0, out1 => #COut.Gen.CoilDiameter)
      wire#w4
      Contact( #CIn.DecoilersHRot.Decoiler1_InLine )
      Move(in := 1, out1 => #COut.Gen.DecoilerInLineNumber)
      Move(in := #CIn.Decoiler1.CoilDiameter, out1 => #COut.Gen.CoilDiameter)
   END_RUNG
   RUNG wire#w4
      Contact( #CIn.DecoilersHRot.Decoiler2_InLine )
      Move(in := 2, out1 => #COut.Gen.DecoilerInLineNumber)
      Move(in := #CIn.Decoiler2.CoilDiameter, out1 => #COut.Gen.CoilDiameter)
   END_RUNG
   // the same network as SCL:
   #COut.Gen.MaterialPresence := ((#Pers.Data.MaterialPresence_StraightenerEntry AND #Pers.Data.MaterialPresence_StraightenerExit) OR #COut.Gen.MaterialPresence) AND #Pers.Data.MaterialPresence_JBPinchExit;
   #COut.Gen.MaterialMissing := NOT #Pers.Data.MaterialPresence_StraightenerEntry AND NOT #Pers.Data.MaterialPresence_StraightenerExit AND NOT #Pers.Data.MaterialPresence_JBPinchExit;
   #COut.Gen.NextEndOfMaterial := #COut.Gen.MaterialPresence AND (NOT #Pers.Data.MaterialPresence_StraightenerEntry OR NOT #Pers.Data.MaterialPresence_StraightenerExit);
   #COut.Gen.EmptyingConfirmed := #COut.Gen.EmptyingConfirmed;
   #COut.Gen.ExtraLowSpeedSelection := #Sts.ExtraLowSpeedSelection;
   #COut.Gen.SemiAutomatic := NOT (NOT #Sts.Semiautomatic AND NOT #TON_Emptying.Q);
   #COut.Gen.Production_Running := NOT (NOT #AreaInterface.Cycle);
   #COut.Gen.DecoilerInLineNumber := 0;
   #COut.Gen.CoilDiameter := 0.0;
   IF #CIn.DecoilersHRot.Decoiler1_InLine THEN
       #COut.Gen.DecoilerInLineNumber := 1;
       #COut.Gen.CoilDiameter := #CIn.Decoiler1.CoilDiameter;
   END_IF;
   IF #CIn.DecoilersHRot.Decoiler2_InLine THEN
       #COut.Gen.DecoilerInLineNumber := 2;
       #COut.Gen.CoilDiameter := #CIn.Decoiler2.CoilDiameter;
   END_IF;
END_REGION

REGION Network 75: <+>
END_REGION

REGION Network 76 (SCL): Coordination Out - Decoiler / Straightener / JB Pinch Roll - Target Velocity
   #COut.Straightener.Feed.Vel := 0.0;

   IF #COut.DecoilerInLine.ModePneumaticBraking THEN
       #COut.DecoilerInLine.Feed.Vel := 0.0;
   END_IF;
   #COut.JB.PinchRoll_Feed.Vel := 0.0;


   IF #Sts.MaterialMoveSemiAut.Bwd_Phase3 THEN

       #Decoiler_VelFactor := 1.0;


       // velocity factor for extralow speed selection
       // 
       IF #Sts.ExtraLowSpeedSelection THEN
           #Decoiler_VelFactor := #Pers.Par.ExtraLowSpeed_Percentage / 100.0;
       END_IF;

       #COut.DecoilerInLine.Feed.Vel := #Pers.Par.SemiAut.Vel_Bkw * #Decoiler_VelFactor;

       #COut.Straightener.Feed.Vel := "Straightener_PERS".PersistentValues.Feed.Man.VelFwdLow;







   ELSIF #Sts.MaterialMoveSemiAut.Bwd_Phase1 OR #Sts.MaterialMoveSemiAut.Bwd_Phase2 THEN

       #COut.Straightener.Feed.Vel := "Straightener_PERS".PersistentValues.Feed.Man.VelFwdLow;
       #COut.DecoilerInLine.Feed.Vel := 0.0;


   ELSIF #Sts.MaterialMoveSemiAut.Fwd_Phase3 THEN

       #Straightener_VelFactor := 1.0;

       // velocity factor for extralow speed selection
       // 
       IF #Sts.ExtraLowSpeedSelection THEN
           #Straightener_VelFactor := #Pers.Par.ExtraLowSpeed_Percentage / 100.0;
       END_IF;
       #COut.Straightener.Feed.Vel := #Pers.Par.SemiAut.Vel_Fwd * #Straightener_VelFactor;


       #Decoiler_VelFactor := 1.0;
       #COut.DecoilerInLine.Feed.Vel := LREAL_TO_REAL(#COut.Straightener.Feed.Vel) * #Decoiler_VelFactor;


   ELSIF #Sts.MaterialMoveSemiAut.Fwd_Phase1 OR #Sts.MaterialMoveSemiAut.Fwd_Phase2 THEN

       #COut.Straightener.Feed.Vel := 0.0;
       #COut.DecoilerInLine.Feed.Vel := 0.0;



   ELSIF #Sts.MaterialMoveAut.Fwd_Phase3 THEN

       //#######################################################
       // VELOCITY OVERRIDE
       //#######################################################

       // Default Override (1..150%) from HMI status page
       // 
       // #OverRide_VelFactor := #Pers.Data.VelocityOverride / 100.0;

       #OverRide_VelFactor := #CIn.Loop.VelocityOverride / 100.0;


       //#######################################################
       // VELOCITY 
       //#######################################################

       #LineVel := #CIn.Downstream.LineVelocity;

       IF #LineVel <= 0.0 THEN
           #LineVel := "PPrf_MAIN".ON_WORK.A01_CoilHandling.MaterialFeeding.Vel;
       END_IF;

       #Straightener_VelFactor := 1.0;
       #COut.Straightener.Feed.Vel := #LineVel * #Straightener_VelFactor * #OverRide_VelFactor;

       #Decoiler_VelFactor := 1.0;
       #COut.DecoilerInLine.Feed.Vel :=  LREAL_TO_REAL(#COut.Straightener.Feed.Vel) * #Decoiler_VelFactor * #OverRide_VelFactor;


   ELSIF #Sts.MaterialMoveAut.Fwd_Phase1 OR #Sts.MaterialMoveAut.Fwd_Phase2 THEN
       #COut.Straightener.Feed.Vel := 0.0;

       IF #COut.DecoilerInLine.ModePneumaticBraking THEN
           #COut.DecoilerInLine.Feed.Vel := 0.0;
       END_IF;


   ELSIF NOT #Sts.EndOfCoil.Idle THEN
       #COut.JB.PinchRoll_Feed.Vel := MIN(IN1 := #Pers.Par.CoilEnd.Vel, IN2 := #CIn.JB.Pinchroll_Feed.MaxVelocity);

       #Straightener_VelFactor := 1.0 - ABS((#Pers.Par.CoilEnd.PercentageStraightener / 100.0));
       #COut.Straightener.Feed.Vel :=#COut.JB.PinchRoll_Feed.Vel * #Straightener_VelFactor;

       #COut.DecoilerInLine.Feed.Vel := #Pers.Par.CoilEnd.Vel;

   END_IF;
END_REGION

REGION Network 77 (SCL): Coordination Out - Decoiler / Straightener / JB Pinch Roll - Target Acc / Dec / jerk
   IF #Ctrl.Semiautomatic_MaterialFwd OR #Ctrl.Semiautomatic_MaterialBkw THEN

       #COut.Straightener.Feed.Acc := #Pers.Par.SemiAut.Acc;
       #COut.Straightener.Feed.Dec := #Pers.Par.SemiAut.Dec;
       #COut.Straightener.Feed.Jerk := #Pers.Par.SemiAut.Jerk;


   ELSIF  NOT #Sts.EndOfCoil.Idle THEN
       #COut.Straightener.Feed.Acc := #Pers.Par.CoilEnd.Acc;
       #COut.Straightener.Feed.Dec := #Pers.Par.CoilEnd.Dec;
       #COut.Straightener.Feed.Jerk := #Pers.Par.CoilEnd.Jerk;


   ELSIF #AreaInterface.Aut THEN
       #COut.Straightener.Feed.Acc := "PPrf_MAIN".ON_WORK.A01_CoilHandling.MaterialFeeding.Acc;
       #COut.Straightener.Feed.Dec := "PPrf_MAIN".ON_WORK.A01_CoilHandling.MaterialFeeding.Dec;
       #COut.Straightener.Feed.Jerk := "PPrf_MAIN".ON_WORK.A01_CoilHandling.MaterialFeeding.Jerk;


       IF NOT #CIn.Downstream.Aut OR #COut.Straightener.Feed.Acc <= 0 OR #COut.Straightener.Feed.Dec <= 0
       THEN
           #COut.Straightener.Feed.Acc := #Pers.Par.SemiAut.Acc;
           #COut.Straightener.Feed.Dec := #Pers.Par.SemiAut.Dec;
           #COut.Straightener.Feed.Jerk := #Pers.Par.SemiAut.Jerk;
       END_IF;


   END_IF;



   #COut.DecoilerInLine.Feed.Acc := #COut.Straightener.Feed.Acc;
   #COut.DecoilerInLine.Feed.Dec := #COut.Straightener.Feed.Dec;

   #COut.JB.PinchRoll_Feed.Acc := #COut.Straightener.Feed.Acc;
   #COut.JB.PinchRoll_Feed.Dec := #COut.Straightener.Feed.Acc;
END_REGION

REGION Network 78: <+>
END_REGION

